   instSignals45Right.signal00 := FALSE;
   instSignals45Right.signal01 := FALSE;
   instSignals45Right.signal02 := FALSE;
   instSignals45Right.signal03 := FALSE;
   instSignals45Right.signal04 := FALSE;
   instSignals45Right.signal05 := FALSE;
   instSignals45Right.signal06 := FALSE;
   instSignals45Right.signal07 := FALSE;
   instSignals45Right.signal08 := FALSE;
   instSignals45Right.signal09 := FALSE;
   instSignals45Right.signal10 := FALSE;
   instSignals45Right.signal11 := FALSE;
   instSignals45Right.signal12 := FALSE;
   instSignals45Right.signal13 := FALSE;
   instSignals45Right.signal14 := FALSE;
   instSignals45Right.signal15 := FALSE;
   instSignals46Left.signal00 := TRUE;
   instSignals46Left.signal01 := TRUE;
   instSignals46Left.signal02 := TRUE;
   instSignals46Left.signal03 := FALSE;
   instSignals46Left.signal04 := FALSE;
   instSignals46Left.signal05 := FALSE;
   instSignals46Left.signal06 := FALSE;
   instSignals46Left.signal07 := FALSE;
   instSignals46Left.signal08 := FALSE;
   instSignals46Left.signal09 := FALSE;
   instSignals46Left.signal10 := FALSE;
   instSignals46Left.signal11 := FALSE;
   instSignals46Left.signal12 := FALSE;
   instSignals46Left.signal13 := FALSE;
   instSignals46Left.signal14 := FALSE;
   instSignals46Left.signal15 := FALSE;
   instSignals46Right.signal00 := FALSE;
   instSignals46Right.signal01 := FALSE;
   instSignals46Right.signal02 := FALSE;
   instSignals46Right.signal03 := FALSE;
   instSignals46Right.signal04 := FALSE;
   instSignals46Right.signal05 := FALSE;
   instSignals46Right.signal06 := FALSE;
   instSignals46Right.signal07 := FALSE;
   instSignals46Right.signal08 := FALSE;
   instSignals46Right.signal09 := FALSE;
   instSignals46Right.signal10 := FALSE;
   instSignals46Right.signal11 := FALSE;
   instSignals46Right.signal12 := FALSE;
   instSignals46Right.signal13 := FALSE;
   instSignals46Right.signal14 := FALSE;
   instSignals46Right.signal15 := FALSE;
   instSignals47Left.signal00 := FALSE;
   instSignals47Left.signal01 := FALSE;
   instSignals47Left.signal02 := FALSE;
   instSignals47Left.signal03 := FALSE;
   instSignals47Left.signal04 := TRUE;
   instSignals47Left.signal05 := FALSE;
   instSignals47Left.signal06 := FALSE;
   instSignals47Left.signal07 := FALSE;
   instSignals47Left.signal08 := FALSE;
   instSignals47Left.signal09 := FALSE;
   instSignals47Left.signal10 := FALSE;
   instSignals47Left.signal11 := FALSE;
   instSignals47Left.signal12 := FALSE;
   instSignals47Left.signal13 := FALSE;
   instSignals47Left.signal14 := FALSE;
   instSignals47Left.signal15 := FALSE;
   instSignals47Right.signal00 := FALSE;
   instSignals47Right.signal01 := FALSE;
   instSignals47Right.signal02 := FALSE;
   instSignals47Right.signal03 := FALSE;
   instSignals47Right.signal04 := FALSE;
   instSignals47Right.signal05 := FALSE;
   instSignals47Right.signal06 := FALSE;
   instSignals47Right.signal07 := FALSE;
   instSignals47Right.signal08 := FALSE;
   instSignals47Right.signal09 := FALSE;
   instSignals47Right.signal10 := FALSE;
   instSignals47Right.signal11 := FALSE;
   instSignals47Right.signal12 := FALSE;
   instSignals47Right.signal13 := FALSE;
   instSignals47Right.signal14 := FALSE;
   instSignals47Right.signal15 := FALSE;
   instSignals48Left.signal00 := FALSE;
   instSignals48Left.signal01 := FALSE;
   instSignals48Left.signal02 := FALSE;
   instSignals48Left.signal03 := FALSE;
   instSignals48Left.signal04 := FALSE;
   instSignals48Left.signal05 := FALSE;
   instSignals48Left.signal06 := FALSE;
   instSignals48Left.signal07 := FALSE;
   instSignals48Left.signal08 := FALSE;
   instSignals48Left.signal09 := FALSE;
   instSignals48Left.signal10 := FALSE;
   instSignals48Left.signal11 := FALSE;
   instSignals48Left.signal12 := FALSE;
   instSignals48Left.signal13 := FALSE;
   instSignals48Left.signal14 := FALSE;
   instSignals48Left.signal15 := FALSE;
   instSignals48Right.signal00 := FALSE;
   instSignals48Right.signal01 := FALSE;
   instSignals48Right.signal02 := FALSE;
   instSignals48Right.signal03 := FALSE;
   instSignals48Right.signal04 := FALSE;
   instSignals48Right.signal05 := FALSE;
   instSignals48Right.signal06 := FALSE;
   instSignals48Right.signal07 := FALSE;
   instSignals48Right.signal08 := FALSE;
   instSignals48Right.signal09 := FALSE;
   instSignals48Right.signal10 := FALSE;
   instSignals48Right.signal11 := FALSE;
   instSignals48Right.signal12 := FALSE;
   instSignals48Right.signal13 := FALSE;
   instSignals48Right.signal14 := FALSE;
   instSignals48Right.signal15 := FALSE;
   instSignals49Left.signal00 := FALSE;
   instSignals49Left.signal01 := FALSE;
   instSignals49Left.signal02 := FALSE;
   instSignals49Left.signal03 := FALSE;
   instSignals49Left.signal04 := FALSE;
   instSignals49Left.signal05 := FALSE;
   instSignals49Left.signal06 := FALSE;
   instSignals49Left.signal07 := FALSE;
   instSignals49Left.signal08 := FALSE;
   instSignals49Left.signal09 := FALSE;
   instSignals49Left.signal10 := FALSE;
   instSignals49Left.signal11 := FALSE;
   instSignals49Left.signal12 := FALSE;
   instSignals49Left.signal13 := FALSE;
   instSignals49Left.signal14 := FALSE;
   instSignals49Left.signal15 := FALSE;
   instSignals49Right.signal00 := FALSE;
   instSignals49Right.signal01 := FALSE;
   instSignals49Right.signal02 := FALSE;
   instSignals49Right.signal03 := FALSE;
   instSignals49Right.signal04 := FALSE;
   instSignals49Right.signal05 := FALSE;
   instSignals49Right.signal06 := FALSE;
   instSignals49Right.signal07 := FALSE;
   instSignals49Right.signal08 := FALSE;
   instSignals49Right.signal09 := FALSE;
   instSignals49Right.signal10 := FALSE;
   instSignals49Right.signal11 := FALSE;
   instSignals49Right.signal12 := FALSE;
   instSignals49Right.signal13 := FALSE;
   instSignals49Right.signal14 := FALSE;
   instSignals49Right.signal15 := FALSE;
   instSignals50Left.signal00 := FALSE;
   instSignals50Left.signal01 := FALSE;
   instSignals50Left.signal02 := FALSE;
   instSignals50Left.signal03 := FALSE;
   instSignals50Left.signal04 := FALSE;
   instSignals50Left.signal05 := FALSE;
   instSignals50Left.signal06 := FALSE;
   instSignals50Left.signal07 := FALSE;
   instSignals50Left.signal08 := FALSE;
   instSignals50Left.signal09 := FALSE;
   instSignals50Left.signal10 := FALSE;
   instSignals50Left.signal11 := FALSE;
   instSignals50Left.signal12 := FALSE;
   instSignals50Left.signal13 := FALSE;
   instSignals50Left.signal14 := FALSE;
   instSignals50Left.signal15 := FALSE;
   instSignals50Right.signal00 := FALSE;
   instSignals50Right.signal01 := FALSE;
   instSignals50Right.signal02 := FALSE;
   instSignals50Right.signal03 := FALSE;
   instSignals50Right.signal04 := FALSE;
   instSignals50Right.signal05 := FALSE;
   instSignals50Right.signal06 := FALSE;
   instSignals50Right.signal07 := FALSE;
   instSignals50Right.signal08 := FALSE;
   instSignals50Right.signal09 := FALSE;
   instSignals50Right.signal10 := FALSE;
   instSignals50Right.signal11 := FALSE;
   instSignals50Right.signal12 := FALSE;
   instSignals50Right.signal13 := FALSE;
   instSignals50Right.signal14 := FALSE;
   instSignals50Right.signal15 := FALSE;
   instSignals51Left.signal00 := FALSE;
   instSignals51Left.signal01 := FALSE;
   instSignals51Left.signal02 := FALSE;
   instSignals51Left.signal03 := FALSE;
   instSignals51Left.signal04 := FALSE;
   instSignals51Left.signal05 := FALSE;
   instSignals51Left.signal06 := FALSE;
   instSignals51Left.signal07 := FALSE;
   instSignals51Left.signal08 := FALSE;
   instSignals51Left.signal09 := FALSE;
   instSignals51Left.signal10 := FALSE;
   instSignals51Left.signal11 := FALSE;
   instSignals51Left.signal12 := FALSE;
   instSignals51Left.signal13 := FALSE;
   instSignals51Left.signal14 := FALSE;
   instSignals51Left.signal15 := FALSE;
   instSignals51Right.signal00 := FALSE;
   instSignals51Right.signal01 := FALSE;
   instSignals51Right.signal02 := FALSE;
   instSignals51Right.signal03 := FALSE;
   instSignals51Right.signal04 := FALSE;
   instSignals51Right.signal05 := FALSE;
   instSignals51Right.signal06 := FALSE;
   instSignals51Right.signal07 := FALSE;
   instSignals51Right.signal08 := FALSE;
   instSignals51Right.signal09 := FALSE;
   instSignals51Right.signal10 := FALSE;
   instSignals51Right.signal11 := FALSE;
   instSignals51Right.signal12 := FALSE;
   instSignals51Right.signal13 := FALSE;
   instSignals51Right.signal14 := FALSE;
   instSignals51Right.signal15 := FALSE;
   instSignals52Left.signal00 := FALSE;
   instSignals52Left.signal01 := FALSE;
   instSignals52Left.signal02 := FALSE;
   instSignals52Left.signal03 := FALSE;
   instSignals52Left.signal04 := FALSE;
   instSignals52Left.signal05 := FALSE;
   instSignals52Left.signal06 := FALSE;
   instSignals52Left.signal07 := FALSE;
   instSignals52Left.signal08 := FALSE;
   instSignals52Left.signal09 := FALSE;
   instSignals52Left.signal10 := FALSE;
   instSignals52Left.signal11 := FALSE;
   instSignals52Left.signal12 := FALSE;
   instSignals52Left.signal13 := FALSE;
   instSignals52Left.signal14 := FALSE;
   instSignals52Left.signal15 := FALSE;
   instSignals52Right.signal00 := FALSE;
   instSignals52Right.signal01 := FALSE;
   instSignals52Right.signal02 := FALSE;
   instSignals52Right.signal03 := FALSE;
   instSignals52Right.signal04 := FALSE;
   instSignals52Right.signal05 := FALSE;
   instSignals52Right.signal06 := FALSE;
   instSignals52Right.signal07 := FALSE;
   instSignals52Right.signal08 := FALSE;
   instSignals52Right.signal09 := FALSE;
   instSignals52Right.signal10 := FALSE;
   instSignals52Right.signal11 := FALSE;
   instSignals52Right.signal12 := FALSE;
   instSignals52Right.signal13 := FALSE;
   instSignals52Right.signal14 := FALSE;
   instSignals52Right.signal15 := FALSE;
   instSignals53Left.signal00 := FALSE;
   instSignals53Left.signal01 := FALSE;
   instSignals53Left.signal02 := FALSE;
   instSignals53Left.signal03 := FALSE;
   instSignals53Left.signal04 := FALSE;
   instSignals53Left.signal05 := FALSE;
   instSignals53Left.signal06 := FALSE;
   instSignals53Left.signal07 := FALSE;
   instSignals53Left.signal08 := FALSE;
   instSignals53Left.signal09 := FALSE;
   instSignals53Left.signal10 := FALSE;
   instSignals53Left.signal11 := FALSE;
   instSignals53Left.signal12 := FALSE;
   instSignals53Left.signal13 := FALSE;
   instSignals53Left.signal14 := FALSE;
   instSignals53Left.signal15 := FALSE;
   instSignals53Right.signal00 := FALSE;
   instSignals53Right.signal01 := FALSE;
   instSignals53Right.signal02 := FALSE;
   instSignals53Right.signal03 := FALSE;
   instSignals53Right.signal04 := FALSE;
   instSignals53Right.signal05 := FALSE;
   instSignals53Right.signal06 := FALSE;
   instSignals53Right.signal07 := FALSE;
   instSignals53Right.signal08 := FALSE;
   instSignals53Right.signal09 := FALSE;
   instSignals53Right.signal10 := FALSE;
   instSignals53Right.signal11 := FALSE;
   instSignals53Right.signal12 := FALSE;
   instSignals53Right.signal13 := FALSE;
   instSignals53Right.signal14 := FALSE;
   instSignals53Right.signal15 := FALSE;
   instSignals54Left.signal00 := FALSE;
   instSignals54Left.signal01 := FALSE;
   instSignals54Left.signal02 := FALSE;
   instSignals54Left.signal03 := FALSE;
   instSignals54Left.signal04 := FALSE;
   instSignals54Left.signal05 := FALSE;
   instSignals54Left.signal06 := FALSE;
   instSignals54Left.signal07 := FALSE;
   instSignals54Left.signal08 := FALSE;
   instSignals54Left.signal09 := FALSE;
   instSignals54Left.signal10 := FALSE;
   instSignals54Left.signal11 := FALSE;
   instSignals54Left.signal12 := FALSE;
   instSignals54Left.signal13 := FALSE;
   instSignals54Left.signal14 := FALSE;
   instSignals54Left.signal15 := FALSE;
   instSignals54Right.signal00 := FALSE;
   instSignals54Right.signal01 := FALSE;
   instSignals54Right.signal02 := FALSE;
   instSignals54Right.signal03 := FALSE;
   instSignals54Right.signal04 := FALSE;
   instSignals54Right.signal05 := FALSE;
   instSignals54Right.signal06 := FALSE;
   instSignals54Right.signal07 := FALSE;
   instSignals54Right.signal08 := FALSE;
   instSignals54Right.signal09 := FALSE;
   instSignals54Right.signal10 := FALSE;
   instSignals54Right.signal11 := FALSE;
   instSignals54Right.signal12 := FALSE;
   instSignals54Right.signal13 := FALSE;
   instSignals54Right.signal14 := FALSE;
   instSignals54Right.signal15 := FALSE;
   instSignals55Left.signal00 := FALSE;
   instSignals55Left.signal01 := FALSE;
   instSignals55Left.signal02 := FALSE;
   instSignals55Left.signal03 := FALSE;
   instSignals55Left.signal04 := FALSE;
   instSignals55Left.signal05 := FALSE;
   instSignals55Left.signal06 := FALSE;
   instSignals55Left.signal07 := FALSE;
   instSignals55Left.signal08 := FALSE;
   instSignals55Left.signal09 := FALSE;
   instSignals55Left.signal10 := FALSE;
   instSignals55Left.signal11 := FALSE;
   instSignals55Left.signal12 := FALSE;
   instSignals55Left.signal13 := FALSE;
   instSignals55Left.signal14 := FALSE;
   instSignals55Left.signal15 := FALSE;
   instSignals55Right.signal00 := FALSE;
   instSignals55Right.signal01 := FALSE;
   instSignals55Right.signal02 := FALSE;
   instSignals55Right.signal03 := FALSE;
   instSignals55Right.signal04 := FALSE;
   instSignals55Right.signal05 := FALSE;
   instSignals55Right.signal06 := FALSE;
   instSignals55Right.signal07 := FALSE;
   instSignals55Right.signal08 := FALSE;
   instSignals55Right.signal09 := FALSE;
   instSignals55Right.signal10 := FALSE;
   instSignals55Right.signal11 := FALSE;
   instSignals55Right.signal12 := FALSE;
   instSignals55Right.signal13 := FALSE;
   instSignals55Right.signal14 := FALSE;
   instSignals55Right.signal15 := FALSE;
   instSignals56Left.signal00 := FALSE;
   instSignals56Left.signal01 := FALSE;
   instSignals56Left.signal02 := FALSE;
   instSignals56Left.signal03 := FALSE;
   instSignals56Left.signal04 := FALSE;
   instSignals56Left.signal05 := FALSE;
   instSignals56Left.signal06 := FALSE;
   instSignals56Left.signal07 := FALSE;
   instSignals56Left.signal08 := FALSE;
   instSignals56Left.signal09 := FALSE;
   instSignals56Left.signal10 := FALSE;
   instSignals56Left.signal11 := FALSE;
   instSignals56Left.signal12 := FALSE;
   instSignals56Left.signal13 := FALSE;
   instSignals56Left.signal14 := FALSE;
   instSignals56Left.signal15 := FALSE;
   instSignals56Right.signal00 := FALSE;
   instSignals56Right.signal01 := FALSE;
   instSignals56Right.signal02 := FALSE;
   instSignals56Right.signal03 := FALSE;
   instSignals56Right.signal04 := FALSE;
   instSignals56Right.signal05 := FALSE;
   instSignals56Right.signal06 := FALSE;
   instSignals56Right.signal07 := FALSE;
   instSignals56Right.signal08 := FALSE;
   instSignals56Right.signal09 := FALSE;
   instSignals56Right.signal10 := FALSE;
   instSignals56Right.signal11 := FALSE;
   instSignals56Right.signal12 := FALSE;
   instSignals56Right.signal13 := FALSE;
   instSignals56Right.signal14 := FALSE;
   instSignals56Right.signal15 := FALSE;
   instSignals57Left.signal00 := FALSE;
   instSignals57Left.signal01 := FALSE;
   instSignals57Left.signal02 := TRUE;
   instSignals57Left.signal03 := FALSE;
   instSignals57Left.signal04 := FALSE;
   instSignals57Left.signal05 := FALSE;
   instSignals57Left.signal06 := FALSE;
   instSignals57Left.signal07 := FALSE;
   instSignals57Left.signal08 := FALSE;
   instSignals57Left.signal09 := FALSE;
   instSignals57Left.signal10 := FALSE;
   instSignals57Left.signal11 := FALSE;
   instSignals57Left.signal12 := FALSE;
   instSignals57Left.signal13 := FALSE;
   instSignals57Left.signal14 := FALSE;
   instSignals57Left.signal15 := FALSE;
   instSignals57Right.signal00 := FALSE;
   instSignals57Right.signal01 := FALSE;
   instSignals57Right.signal02 := FALSE;
   instSignals57Right.signal03 := FALSE;
   instSignals57Right.signal04 := FALSE;
   instSignals57Right.signal05 := FALSE;
   instSignals57Right.signal06 := FALSE;
   instSignals57Right.signal07 := FALSE;
   instSignals57Right.signal08 := FALSE;
   instSignals57Right.signal09 := FALSE;
   instSignals57Right.signal10 := FALSE;
   instSignals57Right.signal11 := FALSE;
   instSignals57Right.signal12 := FALSE;
   instSignals57Right.signal13 := FALSE;
   instSignals57Right.signal14 := FALSE;
   instSignals57Right.signal15 := FALSE;
   instSignals58Left.signal00 := FALSE;
   instSignals58Left.signal01 := TRUE;
   instSignals58Left.signal02 := TRUE;
   instSignals58Left.signal03 := TRUE;
   instSignals58Left.signal04 := TRUE;
   instSignals58Left.signal05 := TRUE;
   instSignals58Left.signal06 := FALSE;
   instSignals58Left.signal07 := FALSE;
   instSignals58Left.signal08 := FALSE;
   instSignals58Left.signal09 := FALSE;
   instSignals58Left.signal10 := FALSE;
   instSignals58Left.signal11 := FALSE;
   instSignals58Left.signal12 := FALSE;
   instSignals58Left.signal13 := FALSE;
   instSignals58Left.signal14 := FALSE;
   instSignals58Left.signal15 := FALSE;
   instSignals58Right.signal00 := FALSE;
   instSignals58Right.signal01 := FALSE;
   instSignals58Right.signal02 := FALSE;
   instSignals58Right.signal03 := FALSE;
   instSignals58Right.signal04 := FALSE;
   instSignals58Right.signal05 := FALSE;
   instSignals58Right.signal06 := FALSE;
   instSignals58Right.signal07 := FALSE;
   instSignals58Right.signal08 := FALSE;
   instSignals58Right.signal09 := FALSE;
   instSignals58Right.signal10 := FALSE;
   instSignals58Right.signal11 := FALSE;
   instSignals58Right.signal12 := FALSE;
   instSignals58Right.signal13 := FALSE;
   instSignals58Right.signal14 := FALSE;
   instSignals58Right.signal15 := FALSE;
   instSignals59Left.signal00 := FALSE;
   instSignals59Left.signal01 := FALSE;
   instSignals59Left.signal02 := FALSE;
   instSignals59Left.signal03 := FALSE;
   instSignals59Left.signal04 := TRUE;
   instSignals59Left.signal05 := FALSE;
   instSignals59Left.signal06 := TRUE;
   instSignals59Left.signal07 := FALSE;
   instSignals59Left.signal08 := FALSE;
   instSignals59Left.signal09 := FALSE;
   instSignals59Left.signal10 := FALSE;
   instSignals59Left.signal11 := FALSE;
   instSignals59Left.signal12 := FALSE;
   instSignals59Left.signal13 := FALSE;
   instSignals59Left.signal14 := FALSE;
   instSignals59Left.signal15 := FALSE;
   instSignals59Right.signal00 := FALSE;
   instSignals59Right.signal01 := FALSE;
   instSignals59Right.signal02 := FALSE;
   instSignals59Right.signal03 := FALSE;
   instSignals59Right.signal04 := FALSE;
   instSignals59Right.signal05 := FALSE;
   instSignals59Right.signal06 := FALSE;
   instSignals59Right.signal07 := FALSE;
   instSignals59Right.signal08 := FALSE;
   instSignals59Right.signal09 := FALSE;
   instSignals59Right.signal10 := FALSE;
   instSignals59Right.signal11 := FALSE;
   instSignals59Right.signal12 := FALSE;
   instSignals59Right.signal13 := FALSE;
   instSignals59Right.signal14 := FALSE;
   instSignals59Right.signal15 := FALSE;
   instSignals60Left.signal00 := TRUE;
   instSignals60Left.signal01 := FALSE;
   instSignals60Left.signal02 := FALSE;
   instSignals60Left.signal03 := FALSE;
   instSignals60Left.signal04 := FALSE;
   instSignals60Left.signal05 := FALSE;
   instSignals60Left.signal06 := FALSE;
   instSignals60Left.signal07 := FALSE;
   instSignals60Left.signal08 := FALSE;
   instSignals60Left.signal09 := FALSE;
   instSignals60Left.signal10 := FALSE;
   instSignals60Left.signal11 := FALSE;
   instSignals60Left.signal12 := FALSE;
   instSignals60Left.signal13 := FALSE;
   instSignals60Left.signal14 := FALSE;
   instSignals60Left.signal15 := FALSE;
   instSignals60Right.signal00 := FALSE;
   instSignals60Right.signal01 := FALSE;
   instSignals60Right.signal02 := FALSE;
   instSignals60Right.signal03 := FALSE;
   instSignals60Right.signal04 := FALSE;
   instSignals60Right.signal05 := FALSE;
   instSignals60Right.signal06 := FALSE;
   instSignals60Right.signal07 := FALSE;
   instSignals60Right.signal08 := FALSE;
   instSignals60Right.signal09 := FALSE;
   instSignals60Right.signal10 := FALSE;
   instSignals60Right.signal11 := FALSE;
   instSignals60Right.signal12 := FALSE;
   instSignals60Right.signal13 := FALSE;
   instSignals60Right.signal14 := FALSE;
   instSignals60Right.signal15 := FALSE;
   instSignals61Left.signal00 := TRUE;
   instSignals61Left.signal01 := FALSE;
   instSignals61Left.signal02 := FALSE;
   instSignals61Left.signal03 := FALSE;
   instSignals61Left.signal04 := FALSE;
   instSignals61Left.signal05 := FALSE;
   instSignals61Left.signal06 := FALSE;
   instSignals61Left.signal07 := FALSE;
   instSignals61Left.signal08 := FALSE;
   instSignals61Left.signal09 := FALSE;
   instSignals61Left.signal10 := FALSE;
   instSignals61Left.signal11 := FALSE;
   instSignals61Left.signal12 := FALSE;
   instSignals61Left.signal13 := FALSE;
   instSignals61Left.signal14 := FALSE;
   instSignals61Left.signal15 := FALSE;
   instSignals61Right.signal00 := FALSE;
   instSignals61Right.signal01 := FALSE;
   instSignals61Right.signal02 := FALSE;
   instSignals61Right.signal03 := FALSE;
   instSignals61Right.signal04 := FALSE;
   instSignals61Right.signal05 := FALSE;
   instSignals61Right.signal06 := FALSE;
   instSignals61Right.signal07 := FALSE;
   instSignals61Right.signal08 := FALSE;
   instSignals61Right.signal09 := FALSE;
   instSignals61Right.signal10 := FALSE;
   instSignals61Right.signal11 := FALSE;
   instSignals61Right.signal12 := FALSE;
   instSignals61Right.signal13 := FALSE;
   instSignals61Right.signal14 := FALSE;
   instSignals61Right.signal15 := FALSE;
   instSignals62Left.signal00 := TRUE;
   instSignals62Left.signal01 := TRUE;
   instSignals62Left.signal02 := TRUE;
   instSignals62Left.signal03 := TRUE;
   instSignals62Left.signal04 := TRUE;
   instSignals62Left.signal05 := TRUE;
   instSignals62Left.signal06 := TRUE;
   instSignals62Left.signal07 := TRUE;
   instSignals62Left.signal08 := FALSE;
   instSignals62Left.signal09 := TRUE;
   instSignals62Left.signal10 := FALSE;
   instSignals62Left.signal11 := TRUE;
   instSignals62Left.signal12 := FALSE;
   instSignals62Left.signal13 := FALSE;
   instSignals62Left.signal14 := FALSE;
   instSignals62Left.signal15 := FALSE;
   instSignals62Right.signal00 := FALSE;
   instSignals62Right.signal01 := FALSE;
   instSignals62Right.signal02 := FALSE;
   instSignals62Right.signal03 := FALSE;
   instSignals62Right.signal04 := FALSE;
   instSignals62Right.signal05 := FALSE;
   instSignals62Right.signal06 := FALSE;
   instSignals62Right.signal07 := FALSE;
   instSignals62Right.signal08 := FALSE;
   instSignals62Right.signal09 := FALSE;
   instSignals62Right.signal10 := FALSE;
   instSignals62Right.signal11 := FALSE;
   instSignals62Right.signal12 := FALSE;
   instSignals62Right.signal13 := FALSE;
   instSignals62Right.signal14 := FALSE;
   instSignals62Right.signal15 := FALSE;
   instSignals63Left.signal00 := TRUE;
   instSignals63Left.signal01 := FALSE;
   instSignals63Left.signal02 := FALSE;
   instSignals63Left.signal03 := FALSE;
   instSignals63Left.signal04 := FALSE;
   instSignals63Left.signal05 := FALSE;
   instSignals63Left.signal06 := FALSE;
   instSignals63Left.signal07 := FALSE;
   instSignals63Left.signal08 := FALSE;
   instSignals63Left.signal09 := FALSE;
   instSignals63Left.signal10 := FALSE;
   instSignals63Left.signal11 := FALSE;
   instSignals63Left.signal12 := FALSE;
   instSignals63Left.signal13 := FALSE;
   instSignals63Left.signal14 := FALSE;
   instSignals63Left.signal15 := FALSE;
   instSignals63Right.signal00 := FALSE;
   instSignals63Right.signal01 := FALSE;
   instSignals63Right.signal02 := FALSE;
   instSignals63Right.signal03 := FALSE;
   instSignals63Right.signal04 := FALSE;
   instSignals63Right.signal05 := FALSE;
   instSignals63Right.signal06 := FALSE;
   instSignals63Right.signal07 := FALSE;
   instSignals63Right.signal08 := FALSE;
   instSignals63Right.signal09 := FALSE;
   instSignals63Right.signal10 := FALSE;
   instSignals63Right.signal11 := FALSE;
   instSignals63Right.signal12 := FALSE;
   instSignals63Right.signal13 := FALSE;
   instSignals63Right.signal14 := FALSE;
   instSignals63Right.signal15 := FALSE;
   instSignals64Left.signal00 := FALSE;
   instSignals64Left.signal01 := FALSE;
   instSignals64Left.signal02 := FALSE;
   instSignals64Left.signal03 := FALSE;
   instSignals64Left.signal04 := FALSE;
   instSignals64Left.signal05 := FALSE;
   instSignals64Left.signal06 := FALSE;
   instSignals64Left.signal07 := FALSE;
   instSignals64Left.signal08 := FALSE;
   instSignals64Left.signal09 := FALSE;
   instSignals64Left.signal10 := FALSE;
   instSignals64Left.signal11 := FALSE;
   instSignals64Left.signal12 := FALSE;
   instSignals64Left.signal13 := FALSE;
   instSignals64Left.signal14 := FALSE;
   instSignals64Left.signal15 := FALSE;
   instSignals64Right.signal00 := FALSE;
   instSignals64Right.signal01 := FALSE;
   instSignals64Right.signal02 := FALSE;
   instSignals64Right.signal03 := FALSE;
   instSignals64Right.signal04 := FALSE;
   instSignals64Right.signal05 := FALSE;
   instSignals64Right.signal06 := FALSE;
   instSignals64Right.signal07 := FALSE;
   instSignals64Right.signal08 := FALSE;
   instSignals64Right.signal09 := FALSE;
   instSignals64Right.signal10 := FALSE;
   instSignals64Right.signal11 := FALSE;
   instSignals64Right.signal12 := FALSE;
   instSignals64Right.signal13 := FALSE;
   instSignals64Right.signal14 := FALSE;
   instSignals64Right.signal15 := FALSE;
   instSignals65Left.signal00 := FALSE;
   instSignals65Left.signal01 := FALSE;
   instSignals65Left.signal02 := FALSE;
   instSignals65Left.signal03 := FALSE;
   instSignals65Left.signal04 := FALSE;
   instSignals65Left.signal05 := FALSE;
   instSignals65Left.signal06 := FALSE;
   instSignals65Left.signal07 := FALSE;
   instSignals65Left.signal08 := FALSE;
   instSignals65Left.signal09 := FALSE;
   instSignals65Left.signal10 := FALSE;
   instSignals65Left.signal11 := FALSE;
   instSignals65Left.signal12 := FALSE;
   instSignals65Left.signal13 := FALSE;
   instSignals65Left.signal14 := FALSE;
   instSignals65Left.signal15 := FALSE;
   instSignals65Right.signal00 := FALSE;
   instSignals65Right.signal01 := FALSE;
   instSignals65Right.signal02 := FALSE;
   instSignals65Right.signal03 := FALSE;
   instSignals65Right.signal04 := FALSE;
   instSignals65Right.signal05 := FALSE;
   instSignals65Right.signal06 := FALSE;
   instSignals65Right.signal07 := FALSE;
   instSignals65Right.signal08 := FALSE;
   instSignals65Right.signal09 := FALSE;
   instSignals65Right.signal10 := FALSE;
   instSignals65Right.signal11 := FALSE;
   instSignals65Right.signal12 := FALSE;
   instSignals65Right.signal13 := FALSE;
   instSignals65Right.signal14 := FALSE;
   instSignals65Right.signal15 := FALSE;
   instSignals66Left.signal00 := FALSE;
   instSignals66Left.signal01 := FALSE;
   instSignals66Left.signal02 := FALSE;
   instSignals66Left.signal03 := FALSE;
   instSignals66Left.signal04 := FALSE;
   instSignals66Left.signal05 := FALSE;
   instSignals66Left.signal06 := FALSE;
   instSignals66Left.signal07 := FALSE;
   instSignals66Left.signal08 := FALSE;
   instSignals66Left.signal09 := FALSE;
   instSignals66Left.signal10 := FALSE;
   instSignals66Left.signal11 := FALSE;
   instSignals66Left.signal12 := FALSE;
   instSignals66Left.signal13 := FALSE;
   instSignals66Left.signal14 := FALSE;
   instSignals66Left.signal15 := FALSE;
   instSignals66Right.signal00 := FALSE;
   instSignals66Right.signal01 := FALSE;
   instSignals66Right.signal02 := FALSE;
   instSignals66Right.signal03 := FALSE;
   instSignals66Right.signal04 := FALSE;
   instSignals66Right.signal05 := FALSE;
   instSignals66Right.signal06 := FALSE;
   instSignals66Right.signal07 := FALSE;
   instSignals66Right.signal08 := FALSE;
   instSignals66Right.signal09 := FALSE;
   instSignals66Right.signal10 := FALSE;
   instSignals66Right.signal11 := FALSE;
   instSignals66Right.signal12 := FALSE;
   instSignals66Right.signal13 := FALSE;
   instSignals66Right.signal14 := FALSE;
   instSignals66Right.signal15 := FALSE;
   instSignals67Left.signal00 := TRUE;
   instSignals67Left.signal01 := FALSE;
   instSignals67Left.signal02 := FALSE;
   instSignals67Left.signal03 := FALSE;
   instSignals67Left.signal04 := FALSE;
   instSignals67Left.signal05 := FALSE;
   instSignals67Left.signal06 := FALSE;
   instSignals67Left.signal07 := FALSE;
   instSignals67Left.signal08 := FALSE;
   instSignals67Left.signal09 := FALSE;
   instSignals67Left.signal10 := FALSE;
   instSignals67Left.signal11 := FALSE;
   instSignals67Left.signal12 := FALSE;
   instSignals67Left.signal13 := FALSE;
   instSignals67Left.signal14 := FALSE;
   instSignals67Left.signal15 := FALSE;
   instSignals67Right.signal00 := FALSE;
   instSignals67Right.signal01 := FALSE;
   instSignals67Right.signal02 := FALSE;
   instSignals67Right.signal03 := FALSE;
   instSignals67Right.signal04 := FALSE;
   instSignals67Right.signal05 := FALSE;
   instSignals67Right.signal06 := FALSE;
   instSignals67Right.signal07 := FALSE;
   instSignals67Right.signal08 := FALSE;
   instSignals67Right.signal09 := FALSE;
   instSignals67Right.signal10 := FALSE;
   instSignals67Right.signal11 := FALSE;
   instSignals67Right.signal12 := FALSE;
   instSignals67Right.signal13 := FALSE;
   instSignals67Right.signal14 := FALSE;
   instSignals67Right.signal15 := FALSE;
   instSignals68Left.signal00 := FALSE;
   instSignals68Left.signal01 := FALSE;
   instSignals68Left.signal02 := FALSE;
   instSignals68Left.signal03 := FALSE;
   instSignals68Left.signal04 := FALSE;
   instSignals68Left.signal05 := FALSE;
   instSignals68Left.signal06 := FALSE;
   instSignals68Left.signal07 := FALSE;
   instSignals68Left.signal08 := FALSE;
   instSignals68Left.signal09 := FALSE;
   instSignals68Left.signal10 := FALSE;
   instSignals68Left.signal11 := FALSE;
   instSignals68Left.signal12 := FALSE;
   instSignals68Left.signal13 := FALSE;
   instSignals68Left.signal14 := FALSE;
   instSignals68Left.signal15 := FALSE;
   instSignals68Right.signal00 := FALSE;
   instSignals68Right.signal01 := FALSE;
   instSignals68Right.signal02 := FALSE;
   instSignals68Right.signal03 := FALSE;
   instSignals68Right.signal04 := FALSE;
   instSignals68Right.signal05 := FALSE;
   instSignals68Right.signal06 := FALSE;
   instSignals68Right.signal07 := FALSE;
   instSignals68Right.signal08 := FALSE;
   instSignals68Right.signal09 := FALSE;
   instSignals68Right.signal10 := FALSE;
   instSignals68Right.signal11 := FALSE;
   instSignals68Right.signal12 := FALSE;
   instSignals68Right.signal13 := FALSE;
   instSignals68Right.signal14 := FALSE;
   instSignals68Right.signal15 := FALSE;
   instSignals69Left.signal00 := FALSE;
   instSignals69Left.signal01 := TRUE;
   instSignals69Left.signal02 := FALSE;
   instSignals69Left.signal03 := FALSE;
   instSignals69Left.signal04 := FALSE;
   instSignals69Left.signal05 := FALSE;
   instSignals69Left.signal06 := FALSE;
   instSignals69Left.signal07 := FALSE;
   instSignals69Left.signal08 := FALSE;
   instSignals69Left.signal09 := FALSE;
   instSignals69Left.signal10 := FALSE;
   instSignals69Left.signal11 := FALSE;
   instSignals69Left.signal12 := FALSE;
   instSignals69Left.signal13 := FALSE;
   instSignals69Left.signal14 := FALSE;
   instSignals69Left.signal15 := FALSE;
   instSignals69Right.signal00 := FALSE;
   instSignals69Right.signal01 := FALSE;
   instSignals69Right.signal02 := FALSE;
   instSignals69Right.signal03 := FALSE;
   instSignals69Right.signal04 := FALSE;
   instSignals69Right.signal05 := FALSE;
   instSignals69Right.signal06 := FALSE;
   instSignals69Right.signal07 := FALSE;
   instSignals69Right.signal08 := FALSE;
   instSignals69Right.signal09 := FALSE;
   instSignals69Right.signal10 := FALSE;
   instSignals69Right.signal11 := FALSE;
   instSignals69Right.signal12 := FALSE;
   instSignals69Right.signal13 := FALSE;
   instSignals69Right.signal14 := FALSE;
   instSignals69Right.signal15 := FALSE;
   instSignals70Left.signal00 := FALSE;
   instSignals70Left.signal01 := FALSE;
   instSignals70Left.signal02 := FALSE;
   instSignals70Left.signal03 := FALSE;
   instSignals70Left.signal04 := FALSE;
   instSignals70Left.signal05 := FALSE;
   instSignals70Left.signal06 := FALSE;
   instSignals70Left.signal07 := FALSE;
   instSignals70Left.signal08 := FALSE;
   instSignals70Left.signal09 := FALSE;
   instSignals70Left.signal10 := FALSE;
   instSignals70Left.signal11 := FALSE;
   instSignals70Left.signal12 := FALSE;
   instSignals70Left.signal13 := FALSE;
   instSignals70Left.signal14 := FALSE;
   instSignals70Left.signal15 := FALSE;
   instSignals70Right.signal00 := FALSE;
   instSignals70Right.signal01 := FALSE;
   instSignals70Right.signal02 := FALSE;
   instSignals70Right.signal03 := FALSE;
   instSignals70Right.signal04 := FALSE;
   instSignals70Right.signal05 := FALSE;
   instSignals70Right.signal06 := FALSE;
   instSignals70Right.signal07 := FALSE;
   instSignals70Right.signal08 := FALSE;
   instSignals70Right.signal09 := FALSE;
   instSignals70Right.signal10 := FALSE;
   instSignals70Right.signal11 := FALSE;
   instSignals70Right.signal12 := FALSE;
   instSignals70Right.signal13 := FALSE;
   instSignals70Right.signal14 := FALSE;
   instSignals70Right.signal15 := FALSE;
   instSignals71Left.signal00 := FALSE;
   instSignals71Left.signal01 := FALSE;
   instSignals71Left.signal02 := FALSE;
   instSignals71Left.signal03 := FALSE;
   instSignals71Left.signal04 := FALSE;
   instSignals71Left.signal05 := FALSE;
   instSignals71Left.signal06 := FALSE;
   instSignals71Left.signal07 := FALSE;
   instSignals71Left.signal08 := FALSE;
   instSignals71Left.signal09 := FALSE;
   instSignals71Left.signal10 := FALSE;
   instSignals71Left.signal11 := FALSE;
   instSignals71Left.signal12 := FALSE;
   instSignals71Left.signal13 := FALSE;
   instSignals71Left.signal14 := FALSE;
   instSignals71Left.signal15 := FALSE;
   instSignals71Right.signal00 := FALSE;
   instSignals71Right.signal01 := FALSE;
   instSignals71Right.signal02 := FALSE;
   instSignals71Right.signal03 := FALSE;
   instSignals71Right.signal04 := FALSE;
   instSignals71Right.signal05 := FALSE;
   instSignals71Right.signal06 := FALSE;
   instSignals71Right.signal07 := FALSE;
   instSignals71Right.signal08 := FALSE;
   instSignals71Right.signal09 := FALSE;
   instSignals71Right.signal10 := FALSE;
   instSignals71Right.signal11 := FALSE;
   instSignals71Right.signal12 := FALSE;
   instSignals71Right.signal13 := FALSE;
   instSignals71Right.signal14 := FALSE;
   instSignals71Right.signal15 := FALSE;
   instSignals72Left.signal00 := FALSE;
   instSignals72Left.signal01 := FALSE;
   instSignals72Left.signal02 := FALSE;
   instSignals72Left.signal03 := FALSE;
   instSignals72Left.signal04 := FALSE;
   instSignals72Left.signal05 := FALSE;
   instSignals72Left.signal06 := FALSE;
   instSignals72Left.signal07 := FALSE;
   instSignals72Left.signal08 := FALSE;
   instSignals72Left.signal09 := FALSE;
   instSignals72Left.signal10 := FALSE;
   instSignals72Left.signal11 := FALSE;
   instSignals72Left.signal12 := FALSE;
   instSignals72Left.signal13 := FALSE;
   instSignals72Left.signal14 := FALSE;
   instSignals72Left.signal15 := FALSE;
   instSignals72Right.signal00 := FALSE;
   instSignals72Right.signal01 := FALSE;
   instSignals72Right.signal02 := FALSE;
   instSignals72Right.signal03 := FALSE;
   instSignals72Right.signal04 := FALSE;
   instSignals72Right.signal05 := FALSE;
   instSignals72Right.signal06 := FALSE;
   instSignals72Right.signal07 := FALSE;
   instSignals72Right.signal08 := FALSE;
   instSignals72Right.signal09 := FALSE;
   instSignals72Right.signal10 := FALSE;
   instSignals72Right.signal11 := FALSE;
   instSignals72Right.signal12 := FALSE;
   instSignals72Right.signal13 := FALSE;
   instSignals72Right.signal14 := FALSE;
   instSignals72Right.signal15 := FALSE;
   instSignals73Left.signal00 := FALSE;
   instSignals73Left.signal01 := FALSE;
   instSignals73Left.signal02 := FALSE;
   instSignals73Left.signal03 := FALSE;
   instSignals73Left.signal04 := FALSE;
   instSignals73Left.signal05 := FALSE;
   instSignals73Left.signal06 := FALSE;
   instSignals73Left.signal07 := FALSE;
   instSignals73Left.signal08 := FALSE;
   instSignals73Left.signal09 := FALSE;
   instSignals73Left.signal10 := FALSE;
   instSignals73Left.signal11 := FALSE;
   instSignals73Left.signal12 := FALSE;
   instSignals73Left.signal13 := FALSE;
   instSignals73Left.signal14 := FALSE;
   instSignals73Left.signal15 := FALSE;
   instSignals73Right.signal00 := FALSE;
   instSignals73Right.signal01 := FALSE;
   instSignals73Right.signal02 := FALSE;
   instSignals73Right.signal03 := FALSE;
   instSignals73Right.signal04 := FALSE;
   instSignals73Right.signal05 := FALSE;
   instSignals73Right.signal06 := FALSE;
   instSignals73Right.signal07 := FALSE;
   instSignals73Right.signal08 := FALSE;
   instSignals73Right.signal09 := FALSE;
   instSignals73Right.signal10 := FALSE;
   instSignals73Right.signal11 := FALSE;
   instSignals73Right.signal12 := FALSE;
   instSignals73Right.signal13 := FALSE;
   instSignals73Right.signal14 := FALSE;
   instSignals73Right.signal15 := FALSE;
   instSignals74Left.signal00 := FALSE;
   instSignals74Left.signal01 := FALSE;
   instSignals74Left.signal02 := FALSE;
   instSignals74Left.signal03 := FALSE;
   instSignals74Left.signal04 := FALSE;
   instSignals74Left.signal05 := FALSE;
   instSignals74Left.signal06 := FALSE;
   instSignals74Left.signal07 := FALSE;
   instSignals74Left.signal08 := FALSE;
   instSignals74Left.signal09 := FALSE;
   instSignals74Left.signal10 := FALSE;
   instSignals74Left.signal11 := FALSE;
   instSignals74Left.signal12 := FALSE;
   instSignals74Left.signal13 := FALSE;
   instSignals74Left.signal14 := FALSE;
   instSignals74Left.signal15 := FALSE;
   instSignals74Right.signal00 := FALSE;
   instSignals74Right.signal01 := FALSE;
   instSignals74Right.signal02 := FALSE;
   instSignals74Right.signal03 := FALSE;
   instSignals74Right.signal04 := FALSE;
   instSignals74Right.signal05 := FALSE;
   instSignals74Right.signal06 := FALSE;
   instSignals74Right.signal07 := FALSE;
   instSignals74Right.signal08 := FALSE;
   instSignals74Right.signal09 := FALSE;
   instSignals74Right.signal10 := FALSE;
   instSignals74Right.signal11 := FALSE;
   instSignals74Right.signal12 := FALSE;
   instSignals74Right.signal13 := FALSE;
   instSignals74Right.signal14 := FALSE;
   instSignals74Right.signal15 := FALSE;
   instSignals75Left.signal00 := FALSE;
   instSignals75Left.signal01 := FALSE;
   instSignals75Left.signal02 := FALSE;
   instSignals75Left.signal03 := FALSE;
   instSignals75Left.signal04 := FALSE;
   instSignals75Left.signal05 := FALSE;
   instSignals75Left.signal06 := FALSE;
   instSignals75Left.signal07 := FALSE;
   instSignals75Left.signal08 := FALSE;
   instSignals75Left.signal09 := FALSE;
   instSignals75Left.signal10 := FALSE;
   instSignals75Left.signal11 := FALSE;
   instSignals75Left.signal12 := FALSE;
   instSignals75Left.signal13 := FALSE;
   instSignals75Left.signal14 := FALSE;
   instSignals75Left.signal15 := FALSE;
   instSignals75Right.signal00 := FALSE;
   instSignals75Right.signal01 := FALSE;
   instSignals75Right.signal02 := FALSE;
   instSignals75Right.signal03 := FALSE;
   instSignals75Right.signal04 := FALSE;
   instSignals75Right.signal05 := FALSE;
   instSignals75Right.signal06 := FALSE;
   instSignals75Right.signal07 := FALSE;
   instSignals75Right.signal08 := FALSE;
   instSignals75Right.signal09 := FALSE;
   instSignals75Right.signal10 := FALSE;
   instSignals75Right.signal11 := FALSE;
   instSignals75Right.signal12 := FALSE;
   instSignals75Right.signal13 := FALSE;
   instSignals75Right.signal14 := FALSE;
   instSignals75Right.signal15 := FALSE;
   instSignals76Left.signal00 := FALSE;
   instSignals76Left.signal01 := FALSE;
   instSignals76Left.signal02 := FALSE;
   instSignals76Left.signal03 := FALSE;
   instSignals76Left.signal04 := FALSE;
   instSignals76Left.signal05 := FALSE;
   instSignals76Left.signal06 := FALSE;
   instSignals76Left.signal07 := FALSE;
   instSignals76Left.signal08 := FALSE;
   instSignals76Left.signal09 := FALSE;
   instSignals76Left.signal10 := FALSE;
   instSignals76Left.signal11 := FALSE;
   instSignals76Left.signal12 := FALSE;
   instSignals76Left.signal13 := FALSE;
   instSignals76Left.signal14 := FALSE;
   instSignals76Left.signal15 := FALSE;
   instSignals76Right.signal00 := FALSE;
   instSignals76Right.signal01 := FALSE;
   instSignals76Right.signal02 := FALSE;
   instSignals76Right.signal03 := FALSE;
   instSignals76Right.signal04 := FALSE;
   instSignals76Right.signal05 := FALSE;
   instSignals76Right.signal06 := FALSE;
   instSignals76Right.signal07 := FALSE;
   instSignals76Right.signal08 := FALSE;
   instSignals76Right.signal09 := FALSE;
   instSignals76Right.signal10 := FALSE;
   instSignals76Right.signal11 := FALSE;
   instSignals76Right.signal12 := FALSE;
   instSignals76Right.signal13 := FALSE;
   instSignals76Right.signal14 := FALSE;
   instSignals76Right.signal15 := FALSE;
   instSignals77Left.signal00 := FALSE;
   instSignals77Left.signal01 := FALSE;
   instSignals77Left.signal02 := FALSE;
   instSignals77Left.signal03 := FALSE;
   instSignals77Left.signal04 := FALSE;
   instSignals77Left.signal05 := FALSE;
   instSignals77Left.signal06 := FALSE;
   instSignals77Left.signal07 := FALSE;
   instSignals77Left.signal08 := FALSE;
   instSignals77Left.signal09 := FALSE;
   instSignals77Left.signal10 := FALSE;
   instSignals77Left.signal11 := FALSE;
   instSignals77Left.signal12 := FALSE;
   instSignals77Left.signal13 := FALSE;
   instSignals77Left.signal14 := FALSE;
   instSignals77Left.signal15 := FALSE;
   instSignals77Right.signal00 := FALSE;
   instSignals77Right.signal01 := FALSE;
   instSignals77Right.signal02 := FALSE;
   instSignals77Right.signal03 := FALSE;
   instSignals77Right.signal04 := FALSE;
   instSignals77Right.signal05 := FALSE;
   instSignals77Right.signal06 := FALSE;
   instSignals77Right.signal07 := FALSE;
   instSignals77Right.signal08 := FALSE;
   instSignals77Right.signal09 := FALSE;
   instSignals77Right.signal10 := FALSE;
   instSignals77Right.signal11 := FALSE;
   instSignals77Right.signal12 := FALSE;
   instSignals77Right.signal13 := FALSE;
   instSignals77Right.signal14 := FALSE;
   instSignals77Right.signal15 := FALSE;
   instSignals78Left.signal00 := FALSE;
   instSignals78Left.signal01 := FALSE;
   instSignals78Left.signal02 := FALSE;
   instSignals78Left.signal03 := FALSE;
   instSignals78Left.signal04 := FALSE;
   instSignals78Left.signal05 := FALSE;
   instSignals78Left.signal06 := FALSE;
   instSignals78Left.signal07 := FALSE;
   instSignals78Left.signal08 := FALSE;
   instSignals78Left.signal09 := FALSE;
   instSignals78Left.signal10 := FALSE;
   instSignals78Left.signal11 := FALSE;
   instSignals78Left.signal12 := FALSE;
   instSignals78Left.signal13 := FALSE;
   instSignals78Left.signal14 := FALSE;
   instSignals78Left.signal15 := FALSE;
   instSignals78Right.signal00 := FALSE;
   instSignals78Right.signal01 := FALSE;
   instSignals78Right.signal02 := FALSE;
   instSignals78Right.signal03 := FALSE;
   instSignals78Right.signal04 := FALSE;
   instSignals78Right.signal05 := FALSE;
   instSignals78Right.signal06 := FALSE;
   instSignals78Right.signal07 := FALSE;
   instSignals78Right.signal08 := FALSE;
   instSignals78Right.signal09 := FALSE;
   instSignals78Right.signal10 := FALSE;
   instSignals78Right.signal11 := FALSE;
   instSignals78Right.signal12 := FALSE;
   instSignals78Right.signal13 := FALSE;
   instSignals78Right.signal14 := FALSE;
   instSignals78Right.signal15 := FALSE;
   instSignals79Left.signal00 := FALSE;
   instSignals79Left.signal01 := FALSE;
   instSignals79Left.signal02 := FALSE;
   instSignals79Left.signal03 := FALSE;
   instSignals79Left.signal04 := FALSE;
   instSignals79Left.signal05 := FALSE;
   instSignals79Left.signal06 := FALSE;
   instSignals79Left.signal07 := FALSE;
   instSignals79Left.signal08 := FALSE;
   instSignals79Left.signal09 := FALSE;
   instSignals79Left.signal10 := FALSE;
   instSignals79Left.signal11 := FALSE;
   instSignals79Left.signal12 := FALSE;
   instSignals79Left.signal13 := FALSE;
   instSignals79Left.signal14 := FALSE;
   instSignals79Left.signal15 := FALSE;
   instSignals79Right.signal00 := FALSE;
   instSignals79Right.signal01 := FALSE;
   instSignals79Right.signal02 := FALSE;
   instSignals79Right.signal03 := FALSE;
   instSignals79Right.signal04 := FALSE;
   instSignals79Right.signal05 := FALSE;
   instSignals79Right.signal06 := FALSE;
   instSignals79Right.signal07 := FALSE;
   instSignals79Right.signal08 := FALSE;
   instSignals79Right.signal09 := FALSE;
   instSignals79Right.signal10 := FALSE;
   instSignals79Right.signal11 := FALSE;
   instSignals79Right.signal12 := FALSE;
   instSignals79Right.signal13 := FALSE;
   instSignals79Right.signal14 := FALSE;
   instSignals79Right.signal15 := FALSE;
   instSignals80Left.signal00 := FALSE;
   instSignals80Left.signal01 := FALSE;
   instSignals80Left.signal02 := FALSE;
   instSignals80Left.signal03 := FALSE;
   instSignals80Left.signal04 := FALSE;
   instSignals80Left.signal05 := FALSE;
   instSignals80Left.signal06 := FALSE;
   instSignals80Left.signal07 := FALSE;
   instSignals80Left.signal08 := FALSE;
   instSignals80Left.signal09 := FALSE;
   instSignals80Left.signal10 := FALSE;
   instSignals80Left.signal11 := FALSE;
   instSignals80Left.signal12 := FALSE;
   instSignals80Left.signal13 := FALSE;
   instSignals80Left.signal14 := FALSE;
   instSignals80Left.signal15 := FALSE;
   instSignals80Right.signal00 := FALSE;
   instSignals80Right.signal01 := FALSE;
   instSignals80Right.signal02 := FALSE;
   instSignals80Right.signal03 := FALSE;
   instSignals80Right.signal04 := FALSE;
   instSignals80Right.signal05 := FALSE;
   instSignals80Right.signal06 := FALSE;
   instSignals80Right.signal07 := FALSE;
   instSignals80Right.signal08 := FALSE;
   instSignals80Right.signal09 := FALSE;
   instSignals80Right.signal10 := FALSE;
   instSignals80Right.signal11 := FALSE;
   instSignals80Right.signal12 := FALSE;
   instSignals80Right.signal13 := FALSE;
   instSignals80Right.signal14 := FALSE;
   instSignals80Right.signal15 := FALSE;
   instSignals81Left.signal00 := FALSE;
   instSignals81Left.signal01 := FALSE;
   instSignals81Left.signal02 := FALSE;
   instSignals81Left.signal03 := FALSE;
   instSignals81Left.signal04 := FALSE;
   instSignals81Left.signal05 := FALSE;
   instSignals81Left.signal06 := FALSE;
   instSignals81Left.signal07 := FALSE;
   instSignals81Left.signal08 := FALSE;
   instSignals81Left.signal09 := FALSE;
   instSignals81Left.signal10 := FALSE;
   instSignals81Left.signal11 := FALSE;
   instSignals81Left.signal12 := FALSE;
   instSignals81Left.signal13 := FALSE;
   instSignals81Left.signal14 := FALSE;
   instSignals81Left.signal15 := FALSE;
   instSignals81Right.signal00 := FALSE;
   instSignals81Right.signal01 := FALSE;
   instSignals81Right.signal02 := FALSE;
   instSignals81Right.signal03 := FALSE;
   instSignals81Right.signal04 := FALSE;
   instSignals81Right.signal05 := FALSE;
   instSignals81Right.signal06 := FALSE;
   instSignals81Right.signal07 := FALSE;
   instSignals81Right.signal08 := FALSE;
   instSignals81Right.signal09 := FALSE;
   instSignals81Right.signal10 := FALSE;
   instSignals81Right.signal11 := FALSE;
   instSignals81Right.signal12 := FALSE;
   instSignals81Right.signal13 := FALSE;
   instSignals81Right.signal14 := FALSE;
   instSignals81Right.signal15 := FALSE;
   instSignals82Left.signal00 := FALSE;
   instSignals82Left.signal01 := FALSE;
   instSignals82Left.signal02 := FALSE;
   instSignals82Left.signal03 := FALSE;
   instSignals82Left.signal04 := FALSE;
   instSignals82Left.signal05 := FALSE;
   instSignals82Left.signal06 := FALSE;
   instSignals82Left.signal07 := FALSE;
   instSignals82Left.signal08 := FALSE;
   instSignals82Left.signal09 := FALSE;
   instSignals82Left.signal10 := FALSE;
   instSignals82Left.signal11 := FALSE;
   instSignals82Left.signal12 := FALSE;
   instSignals82Left.signal13 := FALSE;
   instSignals82Left.signal14 := FALSE;
   instSignals82Left.signal15 := FALSE;
   instSignals82Right.signal00 := FALSE;
   instSignals82Right.signal01 := FALSE;
   instSignals82Right.signal02 := FALSE;
   instSignals82Right.signal03 := FALSE;
   instSignals82Right.signal04 := FALSE;
   instSignals82Right.signal05 := FALSE;
   instSignals82Right.signal06 := FALSE;
   instSignals82Right.signal07 := FALSE;
   instSignals82Right.signal08 := FALSE;
   instSignals82Right.signal09 := FALSE;
   instSignals82Right.signal10 := FALSE;
   instSignals82Right.signal11 := FALSE;
   instSignals82Right.signal12 := FALSE;
   instSignals82Right.signal13 := FALSE;
   instSignals82Right.signal14 := FALSE;
   instSignals82Right.signal15 := FALSE;
   instSignals83Left.signal00 := FALSE;
   instSignals83Left.signal01 := FALSE;
   instSignals83Left.signal02 := FALSE;
   instSignals83Left.signal03 := FALSE;
   instSignals83Left.signal04 := FALSE;
   instSignals83Left.signal05 := FALSE;
   instSignals83Left.signal06 := FALSE;
   instSignals83Left.signal07 := FALSE;
   instSignals83Left.signal08 := FALSE;
   instSignals83Left.signal09 := FALSE;
   instSignals83Left.signal10 := FALSE;
   instSignals83Left.signal11 := FALSE;
   instSignals83Left.signal12 := FALSE;
   instSignals83Left.signal13 := FALSE;
   instSignals83Left.signal14 := FALSE;
   instSignals83Left.signal15 := FALSE;
   instSignals83Right.signal00 := FALSE;
   instSignals83Right.signal01 := FALSE;
   instSignals83Right.signal02 := FALSE;
   instSignals83Right.signal03 := FALSE;
   instSignals83Right.signal04 := FALSE;
   instSignals83Right.signal05 := FALSE;
   instSignals83Right.signal06 := FALSE;
   instSignals83Right.signal07 := FALSE;
   instSignals83Right.signal08 := FALSE;
   instSignals83Right.signal09 := FALSE;
   instSignals83Right.signal10 := FALSE;
   instSignals83Right.signal11 := FALSE;
   instSignals83Right.signal12 := FALSE;
   instSignals83Right.signal13 := FALSE;
   instSignals83Right.signal14 := FALSE;
   instSignals83Right.signal15 := FALSE;
   instSignals84Left.signal00 := FALSE;
   instSignals84Left.signal01 := FALSE;
   instSignals84Left.signal02 := FALSE;
   instSignals84Left.signal03 := FALSE;
   instSignals84Left.signal04 := FALSE;
   instSignals84Left.signal05 := FALSE;
   instSignals84Left.signal06 := FALSE;
   instSignals84Left.signal07 := FALSE;
   instSignals84Left.signal08 := FALSE;
   instSignals84Left.signal09 := FALSE;
   instSignals84Left.signal10 := FALSE;
   instSignals84Left.signal11 := FALSE;
   instSignals84Left.signal12 := FALSE;
   instSignals84Left.signal13 := FALSE;
   instSignals84Left.signal14 := FALSE;
   instSignals84Left.signal15 := FALSE;
   instSignals84Right.signal00 := FALSE;
   instSignals84Right.signal01 := FALSE;
   instSignals84Right.signal02 := FALSE;
   instSignals84Right.signal03 := FALSE;
   instSignals84Right.signal04 := FALSE;
   instSignals84Right.signal05 := FALSE;
   instSignals84Right.signal06 := FALSE;
   instSignals84Right.signal07 := FALSE;
   instSignals84Right.signal08 := FALSE;
   instSignals84Right.signal09 := FALSE;
   instSignals84Right.signal10 := FALSE;
   instSignals84Right.signal11 := FALSE;
   instSignals84Right.signal12 := FALSE;
   instSignals84Right.signal13 := FALSE;
   instSignals84Right.signal14 := FALSE;
   instSignals84Right.signal15 := FALSE;
   instSignals85Left.signal00 := FALSE;
   instSignals85Left.signal01 := FALSE;
   instSignals85Left.signal02 := FALSE;
   instSignals85Left.signal03 := FALSE;
   instSignals85Left.signal04 := FALSE;
   instSignals85Left.signal05 := FALSE;
   instSignals85Left.signal06 := FALSE;
   instSignals85Left.signal07 := FALSE;
   instSignals85Left.signal08 := FALSE;
   instSignals85Left.signal09 := FALSE;
   instSignals85Left.signal10 := FALSE;
   instSignals85Left.signal11 := FALSE;
   instSignals85Left.signal12 := FALSE;
   instSignals85Left.signal13 := FALSE;
   instSignals85Left.signal14 := FALSE;
   instSignals85Left.signal15 := FALSE;
   instSignals85Right.signal00 := FALSE;
   instSignals85Right.signal01 := FALSE;
   instSignals85Right.signal02 := FALSE;
   instSignals85Right.signal03 := FALSE;
   instSignals85Right.signal04 := FALSE;
   instSignals85Right.signal05 := FALSE;
   instSignals85Right.signal06 := FALSE;
   instSignals85Right.signal07 := FALSE;
   instSignals85Right.signal08 := FALSE;
   instSignals85Right.signal09 := FALSE;
   instSignals85Right.signal10 := FALSE;
   instSignals85Right.signal11 := FALSE;
   instSignals85Right.signal12 := FALSE;
   instSignals85Right.signal13 := FALSE;
   instSignals85Right.signal14 := FALSE;
   instSignals85Right.signal15 := FALSE;
   instSignals86Left.signal00 := FALSE;
   instSignals86Left.signal01 := FALSE;
   instSignals86Left.signal02 := FALSE;
   instSignals86Left.signal03 := FALSE;
   instSignals86Left.signal04 := FALSE;
   instSignals86Left.signal05 := FALSE;
   instSignals86Left.signal06 := FALSE;
   instSignals86Left.signal07 := FALSE;
   instSignals86Left.signal08 := FALSE;
   instSignals86Left.signal09 := FALSE;
   instSignals86Left.signal10 := FALSE;
   instSignals86Left.signal11 := FALSE;
   instSignals86Left.signal12 := FALSE;
   instSignals86Left.signal13 := FALSE;
   instSignals86Left.signal14 := FALSE;
   instSignals86Left.signal15 := FALSE;
   instSignals86Right.signal00 := FALSE;
   instSignals86Right.signal01 := FALSE;
   instSignals86Right.signal02 := FALSE;
   instSignals86Right.signal03 := FALSE;
   instSignals86Right.signal04 := FALSE;
   instSignals86Right.signal05 := FALSE;
   instSignals86Right.signal06 := FALSE;
   instSignals86Right.signal07 := FALSE;
   instSignals86Right.signal08 := FALSE;
   instSignals86Right.signal09 := FALSE;
   instSignals86Right.signal10 := FALSE;
   instSignals86Right.signal11 := FALSE;
   instSignals86Right.signal12 := FALSE;
   instSignals86Right.signal13 := FALSE;
   instSignals86Right.signal14 := FALSE;
   instSignals86Right.signal15 := FALSE;
   instSignals87Left.signal00 := FALSE;
   instSignals87Left.signal01 := FALSE;
   instSignals87Left.signal02 := FALSE;
   instSignals87Left.signal03 := FALSE;
   instSignals87Left.signal04 := FALSE;
   instSignals87Left.signal05 := FALSE;
   instSignals87Left.signal06 := FALSE;
   instSignals87Left.signal07 := FALSE;
   instSignals87Left.signal08 := FALSE;
   instSignals87Left.signal09 := FALSE;
   instSignals87Left.signal10 := FALSE;
   instSignals87Left.signal11 := FALSE;
   instSignals87Left.signal12 := FALSE;
   instSignals87Left.signal13 := FALSE;
   instSignals87Left.signal14 := FALSE;
   instSignals87Left.signal15 := FALSE;
   instSignals87Right.signal00 := FALSE;
   instSignals87Right.signal01 := FALSE;
   instSignals87Right.signal02 := FALSE;
   instSignals87Right.signal03 := FALSE;
   instSignals87Right.signal04 := FALSE;
   instSignals87Right.signal05 := FALSE;
   instSignals87Right.signal06 := FALSE;
   instSignals87Right.signal07 := FALSE;
   instSignals87Right.signal08 := FALSE;
   instSignals87Right.signal09 := FALSE;
   instSignals87Right.signal10 := FALSE;
   instSignals87Right.signal11 := FALSE;
   instSignals87Right.signal12 := FALSE;
   instSignals87Right.signal13 := FALSE;
   instSignals87Right.signal14 := FALSE;
   instSignals87Right.signal15 := FALSE;
   instSignals88Left.signal00 := FALSE;
   instSignals88Left.signal01 := FALSE;
   instSignals88Left.signal02 := FALSE;
   instSignals88Left.signal03 := FALSE;
   instSignals88Left.signal04 := FALSE;
   instSignals88Left.signal05 := FALSE;
   instSignals88Left.signal06 := FALSE;
   instSignals88Left.signal07 := FALSE;
   instSignals88Left.signal08 := FALSE;
   instSignals88Left.signal09 := FALSE;
   instSignals88Left.signal10 := FALSE;
   instSignals88Left.signal11 := FALSE;
   instSignals88Left.signal12 := FALSE;
   instSignals88Left.signal13 := FALSE;
   instSignals88Left.signal14 := FALSE;
   instSignals88Left.signal15 := FALSE;
   instSignals88Right.signal00 := FALSE;
   instSignals88Right.signal01 := FALSE;
   instSignals88Right.signal02 := FALSE;
   instSignals88Right.signal03 := FALSE;
   instSignals88Right.signal04 := FALSE;
   instSignals88Right.signal05 := FALSE;
   instSignals88Right.signal06 := FALSE;
   instSignals88Right.signal07 := FALSE;
   instSignals88Right.signal08 := FALSE;
   instSignals88Right.signal09 := FALSE;
   instSignals88Right.signal10 := FALSE;
   instSignals88Right.signal11 := FALSE;
   instSignals88Right.signal12 := FALSE;
   instSignals88Right.signal13 := FALSE;
   instSignals88Right.signal14 := FALSE;
   instSignals88Right.signal15 := FALSE;
   instSignals89Left.signal00 := FALSE;
   instSignals89Left.signal01 := FALSE;
   instSignals89Left.signal02 := FALSE;
   instSignals89Left.signal03 := FALSE;
   instSignals89Left.signal04 := FALSE;
   instSignals89Left.signal05 := FALSE;
   instSignals89Left.signal06 := FALSE;
   instSignals89Left.signal07 := FALSE;
   instSignals89Left.signal08 := FALSE;
   instSignals89Left.signal09 := FALSE;
   instSignals89Left.signal10 := FALSE;
   instSignals89Left.signal11 := FALSE;
   instSignals89Left.signal12 := FALSE;
   instSignals89Left.signal13 := FALSE;
   instSignals89Left.signal14 := FALSE;
   instSignals89Left.signal15 := FALSE;
   instSignals89Right.signal00 := FALSE;
   instSignals89Right.signal01 := FALSE;
   instSignals89Right.signal02 := FALSE;
   instSignals89Right.signal03 := FALSE;
   instSignals89Right.signal04 := FALSE;
   instSignals89Right.signal05 := FALSE;
   instSignals89Right.signal06 := FALSE;
   instSignals89Right.signal07 := FALSE;
   instSignals89Right.signal08 := FALSE;
   instSignals89Right.signal09 := FALSE;
   instSignals89Right.signal10 := FALSE;
   instSignals89Right.signal11 := FALSE;
   instSignals89Right.signal12 := FALSE;
   instSignals89Right.signal13 := FALSE;
   instSignals89Right.signal14 := FALSE;
   instSignals89Right.signal15 := FALSE;
   instSignals90Left.signal00 := FALSE;
   instSignals90Left.signal01 := FALSE;
   instSignals90Left.signal02 := FALSE;
   instSignals90Left.signal03 := FALSE;
   instSignals90Left.signal04 := FALSE;
   instSignals90Left.signal05 := FALSE;
   instSignals90Left.signal06 := FALSE;
   instSignals90Left.signal07 := FALSE;
   instSignals90Left.signal08 := FALSE;
   instSignals90Left.signal09 := FALSE;
   instSignals90Left.signal10 := FALSE;
   instSignals90Left.signal11 := FALSE;
   instSignals90Left.signal12 := FALSE;
   instSignals90Left.signal13 := FALSE;
   instSignals90Left.signal14 := FALSE;
   instSignals90Left.signal15 := FALSE;
   instSignals90Right.signal00 := FALSE;
   instSignals90Right.signal01 := FALSE;
   instSignals90Right.signal02 := FALSE;
   instSignals90Right.signal03 := FALSE;
   instSignals90Right.signal04 := FALSE;
   instSignals90Right.signal05 := FALSE;
   instSignals90Right.signal06 := FALSE;
   instSignals90Right.signal07 := FALSE;
   instSignals90Right.signal08 := FALSE;
   instSignals90Right.signal09 := FALSE;
   instSignals90Right.signal10 := FALSE;
   instSignals90Right.signal11 := FALSE;
   instSignals90Right.signal12 := FALSE;
   instSignals90Right.signal13 := FALSE;
   instSignals90Right.signal14 := FALSE;
   instSignals90Right.signal15 := FALSE;
   instSignals91Left.signal00 := FALSE;
   instSignals91Left.signal01 := FALSE;
   instSignals91Left.signal02 := FALSE;
   instSignals91Left.signal03 := FALSE;
   instSignals91Left.signal04 := FALSE;
   instSignals91Left.signal05 := FALSE;
   instSignals91Left.signal06 := FALSE;
   instSignals91Left.signal07 := FALSE;
   instSignals91Left.signal08 := FALSE;
   instSignals91Left.signal09 := FALSE;
   instSignals91Left.signal10 := FALSE;
   instSignals91Left.signal11 := FALSE;
   instSignals91Left.signal12 := FALSE;
   instSignals91Left.signal13 := FALSE;
   instSignals91Left.signal14 := FALSE;
   instSignals91Left.signal15 := FALSE;
   instSignals91Right.signal00 := FALSE;
   instSignals91Right.signal01 := FALSE;
   instSignals91Right.signal02 := FALSE;
   instSignals91Right.signal03 := FALSE;
   instSignals91Right.signal04 := FALSE;
   instSignals91Right.signal05 := FALSE;
   instSignals91Right.signal06 := FALSE;
   instSignals91Right.signal07 := FALSE;
   instSignals91Right.signal08 := FALSE;
   instSignals91Right.signal09 := FALSE;
   instSignals91Right.signal10 := FALSE;
   instSignals91Right.signal11 := FALSE;
   instSignals91Right.signal12 := FALSE;
   instSignals91Right.signal13 := FALSE;
   instSignals91Right.signal14 := FALSE;
   instSignals91Right.signal15 := FALSE;
   instSignals92Left.signal00 := FALSE;
   instSignals92Left.signal01 := FALSE;
   instSignals92Left.signal02 := FALSE;
   instSignals92Left.signal03 := FALSE;
   instSignals92Left.signal04 := FALSE;
   instSignals92Left.signal05 := FALSE;
   instSignals92Left.signal06 := FALSE;
   instSignals92Left.signal07 := FALSE;
   instSignals92Left.signal08 := FALSE;
   instSignals92Left.signal09 := FALSE;
   instSignals92Left.signal10 := FALSE;
   instSignals92Left.signal11 := FALSE;
   instSignals92Left.signal12 := FALSE;
   instSignals92Left.signal13 := FALSE;
   instSignals92Left.signal14 := FALSE;
   instSignals92Left.signal15 := FALSE;
   instSignals92Right.signal00 := FALSE;
   instSignals92Right.signal01 := FALSE;
   instSignals92Right.signal02 := FALSE;
   instSignals92Right.signal03 := FALSE;
   instSignals92Right.signal04 := FALSE;
   instSignals92Right.signal05 := FALSE;
   instSignals92Right.signal06 := FALSE;
   instSignals92Right.signal07 := FALSE;
   instSignals92Right.signal08 := FALSE;
   instSignals92Right.signal09 := FALSE;
   instSignals92Right.signal10 := FALSE;
   instSignals92Right.signal11 := FALSE;
   instSignals92Right.signal12 := FALSE;
   instSignals92Right.signal13 := FALSE;
   instSignals92Right.signal14 := FALSE;
   instSignals92Right.signal15 := FALSE;
   instSignals93Left.signal00 := FALSE;
   instSignals93Left.signal01 := FALSE;
   instSignals93Left.signal02 := FALSE;
   instSignals93Left.signal03 := FALSE;
   instSignals93Left.signal04 := FALSE;
   instSignals93Left.signal05 := FALSE;
   instSignals93Left.signal06 := FALSE;
   instSignals93Left.signal07 := FALSE;
   instSignals93Left.signal08 := FALSE;
   instSignals93Left.signal09 := FALSE;
   instSignals93Left.signal10 := FALSE;
   instSignals93Left.signal11 := FALSE;
   instSignals93Left.signal12 := FALSE;
   instSignals93Left.signal13 := FALSE;
   instSignals93Left.signal14 := FALSE;
   instSignals93Left.signal15 := FALSE;
   instSignals93Right.signal00 := FALSE;
   instSignals93Right.signal01 := FALSE;
   instSignals93Right.signal02 := FALSE;
   instSignals93Right.signal03 := FALSE;
   instSignals93Right.signal04 := FALSE;
   instSignals93Right.signal05 := FALSE;
   instSignals93Right.signal06 := FALSE;
   instSignals93Right.signal07 := FALSE;
   instSignals93Right.signal08 := FALSE;
   instSignals93Right.signal09 := FALSE;
   instSignals93Right.signal10 := FALSE;
   instSignals93Right.signal11 := FALSE;
   instSignals93Right.signal12 := FALSE;
   instSignals93Right.signal13 := FALSE;
   instSignals93Right.signal14 := FALSE;
   instSignals93Right.signal15 := FALSE;
   instSignals94Left.signal00 := FALSE;
   instSignals94Left.signal01 := FALSE;
   instSignals94Left.signal02 := FALSE;
   instSignals94Left.signal03 := FALSE;
   instSignals94Left.signal04 := FALSE;
   instSignals94Left.signal05 := FALSE;
   instSignals94Left.signal06 := FALSE;
   instSignals94Left.signal07 := FALSE;
   instSignals94Left.signal08 := FALSE;
   instSignals94Left.signal09 := FALSE;
   instSignals94Left.signal10 := FALSE;
   instSignals94Left.signal11 := FALSE;
   instSignals94Left.signal12 := FALSE;
   instSignals94Left.signal13 := FALSE;
   instSignals94Left.signal14 := FALSE;
   instSignals94Left.signal15 := FALSE;
   instSignals94Right.signal00 := FALSE;
   instSignals94Right.signal01 := FALSE;
   instSignals94Right.signal02 := FALSE;
   instSignals94Right.signal03 := FALSE;
   instSignals94Right.signal04 := FALSE;
   instSignals94Right.signal05 := FALSE;
   instSignals94Right.signal06 := FALSE;
   instSignals94Right.signal07 := FALSE;
   instSignals94Right.signal08 := FALSE;
   instSignals94Right.signal09 := FALSE;
   instSignals94Right.signal10 := FALSE;
   instSignals94Right.signal11 := FALSE;
   instSignals94Right.signal12 := FALSE;
   instSignals94Right.signal13 := FALSE;
   instSignals94Right.signal14 := FALSE;
   instSignals94Right.signal15 := FALSE;
   instSignals95Left.signal00 := FALSE;
   instSignals95Left.signal01 := FALSE;
   instSignals95Left.signal02 := FALSE;
   instSignals95Left.signal03 := FALSE;
   instSignals95Left.signal04 := FALSE;
   instSignals95Left.signal05 := FALSE;
   instSignals95Left.signal06 := FALSE;
   instSignals95Left.signal07 := FALSE;
   instSignals95Left.signal08 := FALSE;
   instSignals95Left.signal09 := FALSE;
   instSignals95Left.signal10 := FALSE;
   instSignals95Left.signal11 := FALSE;
   instSignals95Left.signal12 := FALSE;
   instSignals95Left.signal13 := FALSE;
   instSignals95Left.signal14 := FALSE;
   instSignals95Left.signal15 := FALSE;
   instSignals95Right.signal00 := FALSE;
   instSignals95Right.signal01 := FALSE;
   instSignals95Right.signal02 := FALSE;
   instSignals95Right.signal03 := FALSE;
   instSignals95Right.signal04 := FALSE;
   instSignals95Right.signal05 := FALSE;
   instSignals95Right.signal06 := FALSE;
   instSignals95Right.signal07 := FALSE;
   instSignals95Right.signal08 := FALSE;
   instSignals95Right.signal09 := FALSE;
   instSignals95Right.signal10 := FALSE;
   instSignals95Right.signal11 := FALSE;
   instSignals95Right.signal12 := FALSE;
   instSignals95Right.signal13 := FALSE;
   instSignals95Right.signal14 := FALSE;
   instSignals95Right.signal15 := FALSE;
   instSignals96Left.signal00 := FALSE;
   instSignals96Left.signal01 := FALSE;
   instSignals96Left.signal02 := FALSE;
   instSignals96Left.signal03 := FALSE;
   instSignals96Left.signal04 := FALSE;
   instSignals96Left.signal05 := FALSE;
   instSignals96Left.signal06 := FALSE;
   instSignals96Left.signal07 := FALSE;
   instSignals96Left.signal08 := FALSE;
   instSignals96Left.signal09 := FALSE;
   instSignals96Left.signal10 := FALSE;
   instSignals96Left.signal11 := FALSE;
   instSignals96Left.signal12 := FALSE;
   instSignals96Left.signal13 := FALSE;
   instSignals96Left.signal14 := FALSE;
   instSignals96Left.signal15 := FALSE;
   instSignals96Right.signal00 := FALSE;
   instSignals96Right.signal01 := FALSE;
   instSignals96Right.signal02 := FALSE;
   instSignals96Right.signal03 := FALSE;
   instSignals96Right.signal04 := FALSE;
   instSignals96Right.signal05 := FALSE;
   instSignals96Right.signal06 := FALSE;
   instSignals96Right.signal07 := FALSE;
   instSignals96Right.signal08 := FALSE;
   instSignals96Right.signal09 := FALSE;
   instSignals96Right.signal10 := FALSE;
   instSignals96Right.signal11 := FALSE;
   instSignals96Right.signal12 := FALSE;
   instSignals96Right.signal13 := FALSE;
   instSignals96Right.signal14 := FALSE;
   instSignals96Right.signal15 := FALSE;
   instSignals97Left.signal00 := FALSE;
   instSignals97Left.signal01 := FALSE;
   instSignals97Left.signal02 := FALSE;
   instSignals97Left.signal03 := FALSE;
   instSignals97Left.signal04 := FALSE;
   instSignals97Left.signal05 := FALSE;
   instSignals97Left.signal06 := FALSE;
   instSignals97Left.signal07 := FALSE;
   instSignals97Left.signal08 := FALSE;
   instSignals97Left.signal09 := FALSE;
   instSignals97Left.signal10 := FALSE;
   instSignals97Left.signal11 := FALSE;
   instSignals97Left.signal12 := FALSE;
   instSignals97Left.signal13 := FALSE;
   instSignals97Left.signal14 := FALSE;
   instSignals97Left.signal15 := FALSE;
   instSignals97Right.signal00 := FALSE;
   instSignals97Right.signal01 := FALSE;
   instSignals97Right.signal02 := FALSE;
   instSignals97Right.signal03 := FALSE;
   instSignals97Right.signal04 := FALSE;
   instSignals97Right.signal05 := FALSE;
   instSignals97Right.signal06 := FALSE;
   instSignals97Right.signal07 := FALSE;
   instSignals97Right.signal08 := FALSE;
   instSignals97Right.signal09 := FALSE;
   instSignals97Right.signal10 := FALSE;
   instSignals97Right.signal11 := FALSE;
   instSignals97Right.signal12 := FALSE;
   instSignals97Right.signal13 := FALSE;
   instSignals97Right.signal14 := FALSE;
   instSignals97Right.signal15 := FALSE;
   instSignals98Left.signal00 := FALSE;
   instSignals98Left.signal01 := FALSE;
   instSignals98Left.signal02 := FALSE;
   instSignals98Left.signal03 := FALSE;
   instSignals98Left.signal04 := FALSE;
   instSignals98Left.signal05 := FALSE;
   instSignals98Left.signal06 := FALSE;
   instSignals98Left.signal07 := FALSE;
   instSignals98Left.signal08 := FALSE;
   instSignals98Left.signal09 := FALSE;
   instSignals98Left.signal10 := FALSE;
   instSignals98Left.signal11 := FALSE;
   instSignals98Left.signal12 := FALSE;
   instSignals98Left.signal13 := FALSE;
   instSignals98Left.signal14 := FALSE;
   instSignals98Left.signal15 := FALSE;
   instSignals98Right.signal00 := FALSE;
   instSignals98Right.signal01 := FALSE;
   instSignals98Right.signal02 := FALSE;
   instSignals98Right.signal03 := FALSE;
   instSignals98Right.signal04 := FALSE;
   instSignals98Right.signal05 := FALSE;
   instSignals98Right.signal06 := FALSE;
   instSignals98Right.signal07 := FALSE;
   instSignals98Right.signal08 := FALSE;
   instSignals98Right.signal09 := FALSE;
   instSignals98Right.signal10 := FALSE;
   instSignals98Right.signal11 := FALSE;
   instSignals98Right.signal12 := FALSE;
   instSignals98Right.signal13 := FALSE;
   instSignals98Right.signal14 := FALSE;
   instSignals98Right.signal15 := FALSE;
   instSignals99Left.signal00 := FALSE;
   instSignals99Left.signal01 := FALSE;
   instSignals99Left.signal02 := FALSE;
   instSignals99Left.signal03 := FALSE;
   instSignals99Left.signal04 := FALSE;
   instSignals99Left.signal05 := FALSE;
   instSignals99Left.signal06 := FALSE;
   instSignals99Left.signal07 := FALSE;
   instSignals99Left.signal08 := FALSE;
   instSignals99Left.signal09 := FALSE;
   instSignals99Left.signal10 := FALSE;
   instSignals99Left.signal11 := FALSE;
   instSignals99Left.signal12 := FALSE;
   instSignals99Left.signal13 := FALSE;
   instSignals99Left.signal14 := FALSE;
   instSignals99Left.signal15 := FALSE;
   instSignals99Right.signal00 := FALSE;
   instSignals99Right.signal01 := FALSE;
   instSignals99Right.signal02 := FALSE;
   instSignals99Right.signal03 := FALSE;
   instSignals99Right.signal04 := FALSE;
   instSignals99Right.signal05 := FALSE;
   instSignals99Right.signal06 := FALSE;
   instSignals99Right.signal07 := FALSE;
   instSignals99Right.signal08 := FALSE;
   instSignals99Right.signal09 := FALSE;
   instSignals99Right.signal10 := FALSE;
   instSignals99Right.signal11 := FALSE;
   instSignals99Right.signal12 := FALSE;
   instSignals99Right.signal13 := FALSE;
   instSignals99Right.signal14 := FALSE;
   instSignals99Right.signal15 := FALSE;
END_DATA_BLOCK

DATA_BLOCK "InstProfinetDeviceDiagStatus"   // DB215
// stored: InstanceOfName LER_DiagnosticsStatus, InstanceOfType FB
"LER_DiagnosticsStatus"
   // VAR_INPUT
   //    devStateHmi_X1 : Array[0..256] of "LAF_typeDevDiagBasic";
   //    devStateHmi_X2 : Array[0..256] of "LAF_typeDevDiagBasic";
   //    UnitSelect : Int := 3;
   //    Reset : Bool := FALSE;
   // END_VAR
   // VAR_IN_OUT
   //    DevState : "LER_DiagnosticsInterface";
   // END_VAR
   // VAR
   //    staticCntState : Int := 189;
   //    staticCntStartState : Int := 1;
   //    staticCntEndState : Int := 200;
   //    staticCntDev : Int := 5;
   //    staticCntHighLimit_X2 : Array[1..15] of Int;
   //    staticCntLowLimit_X2 : Array[1..15] of Int;
   //    staticCntHighLimit_X1 : Array[1..15] of Int;
   //    staticCntLowLimit_X1 : Array[1..15] of Int;
   //    staticCntModuleState : Int := 69;
   //    staticDevStateError : Array[0..15] of Bool;
   //    statiDevStateMove_X1 : Array[0..15] of Int;
   //    statiDevStateMove_X2 : Array[0..15] of Int;
   // END_VAR
BEGIN
   devStateHmi_X1[0..256].devNumber := 0;
   devStateHmi_X1[0..256].devName := '';
   devStateHmi_X1[0..256].devStateDezCoded := 0;
   devStateHmi_X1[0..256].devStateBitCoded := 16#0000;
   devStateHmi_X1[0..256].first8CharOfMlfb := '';
   devStateHmi_X2[0..256].devNumber := 0;
   devStateHmi_X2[0..256].devName := '';
   devStateHmi_X2[0..256].devStateDezCoded := 0;
   devStateHmi_X2[0..256].devStateBitCoded := 16#0000;
   devStateHmi_X2[0..256].first8CharOfMlfb := '';
   staticCntHighLimit_X2[1] := 2;
   staticCntHighLimit_X2[2] := 33;
   staticCntHighLimit_X2[3] := 42;
   staticCntHighLimit_X2[4] := 68;
   staticCntHighLimit_X2[5] := 91;
   staticCntHighLimit_X2[6] := 115;
   staticCntHighLimit_X2[7] := 133;
   staticCntHighLimit_X2[8] := 143;
   staticCntHighLimit_X2[9] := 170;
   staticCntHighLimit_X2[10..15] := 0;
   staticCntLowLimit_X2[1] := 2;
   staticCntLowLimit_X2[2] := 30;
   staticCntLowLimit_X2[3] := 42;
   staticCntLowLimit_X2[4] := 61;
   staticCntLowLimit_X2[5] := 81;
   staticCntLowLimit_X2[6] := 101;
   staticCntLowLimit_X2[7] := 121;
   staticCntLowLimit_X2[8] := 141;
   staticCntLowLimit_X2[9] := 161;
   staticCntLowLimit_X2[10..15] := 0;
   staticCntHighLimit_X1[1] := 1;
   staticCntHighLimit_X1[2] := 29;
   staticCntHighLimit_X1[3] := 41;
   staticCntHighLimit_X1[4..15] := 0;
   staticCntLowLimit_X1[1] := 1;
   staticCntLowLimit_X1[2] := 21;
   staticCntLowLimit_X1[3] := 41;
   staticCntLowLimit_X1[4..15] := 0;
   staticDevStateError[0..15] := FALSE;
   statiDevStateMove_X1[0] := 0;
   statiDevStateMove_X1[1] := 1;
   statiDevStateMove_X1[2] := 9;
   statiDevStateMove_X1[3] := 1;
   statiDevStateMove_X1[4..15] := 0;
   statiDevStateMove_X2[0] := 0;
   statiDevStateMove_X2[1] := 2;
   statiDevStateMove_X2[2] := 13;
   statiDevStateMove_X2[3] := 2;
   statiDevStateMove_X2[4] := 8;
   statiDevStateMove_X2[5] := 11;
   statiDevStateMove_X2[6] := 15;
   statiDevStateMove_X2[7] := 13;
   statiDevStateMove_X2[8] := 3;
   statiDevStateMove_X2[9] := 10;
   statiDevStateMove_X2[10..15] := 0;
END_DATA_BLOCK

DATA_BLOCK "InstProfinetDeviceDiag_x1"   // DB36
AUTHOR : Siemens Digital Industries
FAMILY : LAF
// stored: AssignedProDiagFB ProDiag, InstanceOfName LAF_ProfinetDevDiag, InstanceOfType FB
"LAF_ProfinetDevDiag"
   // VAR_INPUT
   //    plantIdentifier { ExternalAccessible := 'False'; ExternalVisible := 'False'; ExternalWritable := 'False'} : WString[24] := WSTRING#'';
   //    textListId { ExternalAccessible := 'False'; ExternalVisible := 'False'; ExternalWritable := 'False'} : Int := 0;
   //    localProfinetSystem { ExternalAccessible := 'False'; ExternalVisible := 'False'; ExternalWritable := 'False'} : HW_IOSYSTEM := 0;
   //    firstCycle { ExternalAccessible := 'False'; ExternalVisible := 'False'; ExternalWritable := 'False'} : Bool := FALSE;
   //    maxDevicesDiag { ExternalAccessible := 'False'; ExternalVisible := 'False'; ExternalWritable := 'False'} : DInt := 0;
   //    maxModulesDiag { ExternalAccessible := 'False'; ExternalVisible := 'False'; ExternalWritable := 'False'} : DInt := 0;
   //    ackAlarms { ExternalAccessible := 'False'; ExternalVisible := 'False'; ExternalWritable := 'False'} : Bool := FALSE;
   //    hideAlarmMask { ExternalAccessible := 'False'; ExternalVisible := 'False'; ExternalWritable := 'False'} : Word := 16#0000;
   // END_VAR
   // VAR_OUTPUT
   //    generalAlarm { ExternalAccessible := 'False'; ExternalVisible := 'False'; ExternalWritable := 'False'} : Bool := FALSE;
   //    deviceFaulty { ExternalAccessible := 'False'; ExternalVisible := 'False'; ExternalWritable := 'False'} : Bool := FALSE;
   //    deviceProblem { ExternalAccessible := 'False'; ExternalVisible := 'False'; ExternalWritable := 'False'} : Bool := FALSE;
   //    deviceDeactivated { ExternalAccessible := 'False'; ExternalVisible := 'False'; ExternalWritable := 'False'} : Bool := FALSE;
   //    deviceNotPresent { ExternalAccessible := 'False'; ExternalVisible := 'False'; ExternalWritable := 'False'} : Bool := FALSE;
   // END_VAR
   // VAR_IN_OUT
   //    interfaceDevDiag : "LAF_typeDevDiagInterface";
   // END_VAR
   // VAR
   //    statDevDiagInternal { ExternalAccessible := 'False'; ExternalVisible := 'False'; ExternalWritable := 'False'} : "LAF_typeDevDiagInternal";
   //    statCnt1ShotGetName { ExternalAccessible := 'False'; ExternalVisible := 'False'; ExternalWritable := 'False'} : DInt := 1;
   //    statCnt1ShotGeo2Log { ExternalAccessible := 'False'; ExternalVisible := 'False'; ExternalWritable := 'False'} : DInt := 1;
   //    statCnt1ShotGetImDat { ExternalAccessible := 'False'; ExternalVisible := 'False'; ExternalWritable := 'False'} : DInt := 1;
   //    statCntCyclDevState { ExternalAccessible := 'False'; ExternalVisible := 'False'; ExternalWritable := 'False'} : DInt := 1;
   //    statCntCyclState { ExternalAccessible := 'False'; ExternalVisible := 'False'; ExternalWritable := 'False'} : DInt := 1;
   //    statCntCyclModulState { ExternalAccessible := 'False'; ExternalVisible := 'False'; ExternalWritable := 'False'} : DInt := 1;
   //    statCntCyclGetDiag { ExternalAccessible := 'False'; ExternalVisible := 'False'; ExternalWritable := 'False'} : DInt := 1;
   //    statBusy { ExternalAccessible := 'False'; ExternalVisible := 'False'; ExternalWritable := 'False'} : "LAF_typeDevDiagStateInstruct";
   //    statDone { ExternalAccessible := 'False'; ExternalVisible := 'False'; ExternalWritable := 'False'} : "LAF_typeDevDiagStateInstruct";
   //    statOtherInstruct { ExternalAccessible := 'False'; ExternalVisible := 'False'; ExternalWritable := 'False'} : "LAF_typeDevDiagInstruct";
   //    instGetName { ExternalAccessible := 'False'; ExternalVisible := 'False'; ExternalWritable := 'False'} : Get_Name;
   //    statGetNameDat { ExternalAccessible := 'False'; ExternalVisible := 'False'; ExternalWritable := 'False'} : String[24] := '';
   //    statGetNameErrorStatus { ExternalAccessible := 'False'; ExternalVisible := 'False'; ExternalWritable := 'False'} : Word := 16#0000;
   //    statGetNameErrorDevCycle { ExternalAccessible := 'False'; ExternalVisible := 'False'; ExternalWritable := 'False'} : DInt := 0;
   //    instGetImData { ExternalAccessible := 'False'; ExternalVisible := 'False'; ExternalWritable := 'False'} : Get_IM_Data;
   //    statIm0Data { ExternalAccessible := 'False'; ExternalVisible := 'False'; ExternalWritable := 'False'} : IM0_Data;
   //    statGetImDatErrorStatus { ExternalAccessible := 'False'; ExternalVisible := 'False'; ExternalWritable := 'False'} : Word := 16#0000;
   //    statGetImDatErrorCycle { ExternalAccessible := 'False'; ExternalVisible := 'False'; ExternalWritable := 'False'} : DInt := 0;
   //    statAlarm { ExternalAccessible := 'False'; ExternalVisible := 'False'; ExternalWritable := 'False'} : "LAF_typeDevDiagAlarm";
   //    statHideAlarm { ExternalAccessible := 'False'; ExternalVisible := 'False'; ExternalWritable := 'False'} : "LAF_typeDevDiagAlarm";
   //    statRisPushbutton { ExternalAccessible := 'False'; ExternalVisible := 'False'; ExternalWritable := 'False'} : "LAF_typeDevDiagRisEdge";
   //    statErrorText { ExternalAccessible := 'False'; ExternalVisible := 'False'; ExternalWritable := 'False'} : String[24] := 'No Device Name readable';
   //    stat8CharError { ExternalAccessible := 'False'; ExternalVisible := 'False'; ExternalWritable := 'False'} : String[8] := '????????';
   //    statAlarmNo { ExternalAccessible := 'False'; ExternalVisible := 'False'; ExternalWritable := 'False'} : Array[0..23] of UInt;
   // END_VAR
BEGIN
   statDevDiagInternal.localProfinetSystem := 0;
   statDevDiagInternal.maxDevices := 0;
   statDevDiagInternal.maxModules := 0;
   statDevDiagInternal.numberDevices.configured := 0;
   statDevDiagInternal.numberDevices.notPresent := 0;
   statDevDiagInternal.numberDevices.deactivated := 0;
   statDevDiagInternal.numberDevices.faulty := 0;
   statDevDiagInternal.numberDevices.problem := 0;
   statDevDiagInternal.hwAddress[0..256].hwtype2 := 0;
   statDevDiagInternal.hwAddress[0..256].hwtype5 := 0;
   statDevDiagInternal.hwAddress[0..256].hwtype5If := 0;
   statBusy.getName := FALSE;
   statBusy.geo2Log := FALSE;
   statBusy.moduleStates := FALSE;
   statBusy.getDiag := FALSE;
   statBusy.getImData := FALSE;
   statDone.getName := FALSE;
   statDone.geo2Log := FALSE;
   statDone.moduleStates := FALSE;
   statDone.getDiag := FALSE;
   statDone.getImData := FALSE;
   statOtherInstruct.log2GeoLaddr := 0;
   statOtherInstruct.log2GeoRetVal := 0;
   statOtherInstruct.log2Geo.HWTYPE := 0;
   statOtherInstruct.log2Geo.AREA := 0;
   statOtherInstruct.log2Geo.IOSYSTEM := 0;
   statOtherInstruct.log2Geo.STATION := 0;
   statOtherInstruct.log2Geo.SLOT := 0;
   statOtherInstruct.log2Geo.SUBSLOT := 0;
   statOtherInstruct.devStateMode1.laddr := 0;
   statOtherInstruct.devStateMode1.mode := 0;
   statOtherInstruct.devStateMode1.retVal := 0;
   statOtherInstruct.devStateMode1.state[0..1024] := FALSE;
   statOtherInstruct.devStateMode2.laddr := 0;
   statOtherInstruct.devStateMode2.mode := 0;
   statOtherInstruct.devStateMode2.retVal := 0;
   statOtherInstruct.devStateMode2.state[0..1024] := FALSE;
   statOtherInstruct.devStateMode3.laddr := 0;
   statOtherInstruct.devStateMode3.mode := 0;
   statOtherInstruct.devStateMode3.retVal := 0;
   statOtherInstruct.devStateMode3.state[0..1024] := FALSE;
   statOtherInstruct.devStateMode4.laddr := 0;
   statOtherInstruct.devStateMode4.mode := 0;
   statOtherInstruct.devStateMode4.retVal := 0;
   statOtherInstruct.devStateMode4.state[0..1024] := FALSE;
   statOtherInstruct.devStateMode5.laddr := 0;
   statOtherInstruct.devStateMode5.mode := 0;
   statOtherInstruct.devStateMode5.retVal := 0;
   statOtherInstruct.devStateMode5.state[0..1024] := FALSE;
   statOtherInstruct.geo2LogLaddr := 0;
   statOtherInstruct.geo2LogRetVal := 0;
   statOtherInstruct.geo2Log.HWTYPE := 0;
   statOtherInstruct.geo2Log.AREA := 0;
   statOtherInstruct.geo2Log.IOSYSTEM := 0;
   statOtherInstruct.geo2Log.STATION := 0;
   statOtherInstruct.geo2Log.SLOT := 0;
   statOtherInstruct.geo2Log.SUBSLOT := 0;
   statOtherInstruct.moduleStateMode2.laddr := 0;
   statOtherInstruct.moduleStateMode2.mode := 0;
   statOtherInstruct.moduleStateMode2.retVal := 0;
   statOtherInstruct.moduleStateMode2.state[0..127] := FALSE;
   statOtherInstruct.moduleStateMode5.laddr := 0;
   statOtherInstruct.moduleStateMode5.mode := 0;
   statOtherInstruct.moduleStateMode5.retVal := 0;
   statOtherInstruct.moduleStateMode5.state[0..127] := FALSE;
   statOtherInstruct.getDiag.mode := 0;
   statOtherInstruct.getDiag.laddr := 0;
   statOtherInstruct.getDiag.retVal := 0;
   statOtherInstruct.getDiag.cntDiag := 0;
   statOtherInstruct.getDiag.diagDataMode0 := 16#0000_0000;
   statOtherInstruct.getDiag.diagDataMode1.MaintainanceState := 16#0000_0000;
   statOtherInstruct.getDiag.diagDataMode1.ComponentStateDetail := 16#0000_0000;
   statOtherInstruct.getDiag.diagDataMode1.OwnState := 0;
   statOtherInstruct.getDiag.diagDataMode1.IOState := 16#0000;
   statOtherInstruct.getDiag.diagDataMode1.OperatingState := 0;
   statOtherInstruct.getDiag.diagDataMode2.SubordinateState := 0;
   statOtherInstruct.getDiag.diagDataMode2.SubordinateIOState := 16#0000;
   statOtherInstruct.getDiag.diagDataMode2.DNNmode := 16#0000;
   statOtherInstruct.getDiag.detailData := 0;
   instGetName.LADDR := 0;
   instGetName.STATION_NR := 0;
   instGetName.DONE := FALSE;
   instGetName.BUSY := FALSE;
   instGetName.ERROR := FALSE;
   instGetName.LEN := 0;
   instGetName.STATUS := 16#0000;
   instGetName.BusyState := 16#0000;
   instGetImData.LADDR := 0;
   instGetImData.IM_TYPE := 0;
   instGetImData.DONE := FALSE;
   instGetImData.BUSY := FALSE;
   instGetImData.ERROR := FALSE;
   instGetImData.STATUS := 16#0000;
   instGetImData.sdw_GetAttrID := 16#0000_0000;
   instGetImData.sdw_GetAttrAID := 16#0000_0000;
   instGetImData.sdi_SfcLen := 0;
   instGetImData.sb_useGetMultiAttr := FALSE;
   instGetImData.sui_GetMultiAttrACount := 0;
   instGetImData.sa_GetMultiAttrPathLens[0] := 0;
   instGetImData.sa_GetMultiAttrPaths[0..2] := 0;
   instGetImData.sa_GetMultiAttrResultLens[0] := 0;
   instGetImData.sa_GetMultiAttrResult := '';
   instGetImData.sb_SfcValid := FALSE;
   instGetImData.sb_SfcERROR := FALSE;
   instGetImData.sw_SfcStatus := 16#0000;
   instGetImData.sa_SfcData[0..64] := 16#00;
   instGetImData.sudi_arraylength := 0;
   instGetImData.sudi_datatype := 0;
   instGetImData.sui_imdataLen := 0;
   instGetImData.sui_imdataLen_netto := 54;
   instGetImData.si_index := 0;
   instGetImData.sb_SfcLocked := FALSE;
   instGetImData.pw_TemporaryWord := 16#0000;
   instGetImData.pa_DataByte[0..53] := 16#00;
   instGetImData.pa_DataChar[0..53] := ' ';
   instGetImData.pa_TemporaryCharArray[0..19] := ' ';
   instGetImData.p_DataUDT.Manufacturer_ID := 0;
   instGetImData.p_DataUDT.Order_ID := '';
   instGetImData.p_DataUDT.Serial_Number := '';
   instGetImData.p_DataUDT.Hardware_Revision := 0;
   instGetImData.p_DataUDT.Software_Revision."Type" := ' ';
   instGetImData.p_DataUDT.Software_Revision.Functional := 0;
   instGetImData.p_DataUDT.Software_Revision.Bugfix := 0;
   instGetImData.p_DataUDT.Software_Revision.Internal := 0;
   instGetImData.p_DataUDT.Revision_Counter := 0;
   instGetImData.p_DataUDT.Profile_ID := 0;
   instGetImData.p_DataUDT.Profile_Specific_Type := 0;
   instGetImData.p_DataUDT.IM_Version := 16#0000;
   instGetImData.p_DataUDT.IM_Supported := 16#0000;
   statIm0Data.Manufacturer_ID := 0;
   statIm0Data.Order_ID := '';
   statIm0Data.Serial_Number := '';
   statIm0Data.Hardware_Revision := 0;
   statIm0Data.Software_Revision."Type" := ' ';
   statIm0Data.Software_Revision.Functional := 0;
   statIm0Data.Software_Revision.Bugfix := 0;
   statIm0Data.Software_Revision.Internal := 0;
   statIm0Data.Revision_Counter := 0;
   statIm0Data.Profile_ID := 0;
   statIm0Data.Profile_Specific_Type := 0;
   statIm0Data.IM_Version := 16#0000;
   statIm0Data.IM_Supported := 16#0000;
   statAlarm.invalidValueMaxDevices := FALSE;
   statAlarm.invalidValueMaxModules := FALSE;
   statAlarm.invalidAddressLog2Geo := FALSE;
   statAlarm.errorReadDeviceStates := FALSE;
   statAlarm.deviceFaulty := FALSE;
   statAlarm.deviceProblem := FALSE;
   statAlarm.deviceDeactivated := FALSE;
   statAlarm.deviceNotPresent := FALSE;
   statAlarm.deviceNetworkError := FALSE;
   statAlarm.deviceMaintRequired := FALSE;
   statAlarm.deviceMaintDemanded := FALSE;
   statAlarm.spare11 := FALSE;
   statAlarm.spare12 := FALSE;
   statAlarm.spare13 := FALSE;
   statAlarm.spare14 := FALSE;
   statAlarm.spare15 := FALSE;
   statHideAlarm.invalidValueMaxDevices := FALSE;
   statHideAlarm.invalidValueMaxModules := FALSE;
   statHideAlarm.invalidAddressLog2Geo := FALSE;
   statHideAlarm.errorReadDeviceStates := FALSE;
   statHideAlarm.deviceFaulty := FALSE;
   statHideAlarm.deviceProblem := FALSE;
   statHideAlarm.deviceDeactivated := FALSE;
   statHideAlarm.deviceNotPresent := FALSE;
   statHideAlarm.deviceNetworkError := FALSE;
   statHideAlarm.deviceMaintRequired := FALSE;
   statHideAlarm.deviceMaintDemanded := FALSE;
   statHideAlarm.spare11 := FALSE;
   statHideAlarm.spare12 := FALSE;
   statHideAlarm.spare13 := FALSE;
   statHideAlarm.spare14 := FALSE;
   statHideAlarm.spare15 := FALSE;
   statRisPushbutton.risEdgeManualReadAll := FALSE;
   statRisPushbutton.posPulseManualReadAll := FALSE;
   statRisPushbutton.risEdgeResetAll := FALSE;
   statRisPushbutton.posPulseResetAll := FALSE;
   statRisPushbutton.risEdgeQuitAlarms := FALSE;
   statRisPushbutton.posPulseQuitAlarms := FALSE;
   statAlarmNo[0] := 0;
   statAlarmNo[1] := 1;
   statAlarmNo[2] := 2;
   statAlarmNo[3] := 3;
   statAlarmNo[4] := 4;
   statAlarmNo[5] := 5;
   statAlarmNo[6] := 6;
   statAlarmNo[7] := 7;
   statAlarmNo[8] := 8;
   statAlarmNo[9] := 9;
   statAlarmNo[10] := 10;
   statAlarmNo[11] := 11;
   statAlarmNo[12] := 12;
   statAlarmNo[13] := 13;
   statAlarmNo[14] := 14;
   statAlarmNo[15] := 15;
   statAlarmNo[16] := 16;
   statAlarmNo[17] := 17;
   statAlarmNo[18] := 18;
   statAlarmNo[19] := 19;
   statAlarmNo[20] := 20;
   statAlarmNo[21] := 21;
   statAlarmNo[22] := 22;
   statAlarmNo[23] := 23;
END_DATA_BLOCK

